LIN {X 0,Y 129.211,Z 756.744,A -85,B 0,C 180,E1 22949.999,E2 22949.999} C_VEL
LIN {X 0,Y 129.325,Z 753.398,A -85,B 0,C 180,E1 22963.541,E2 22963.541} C_VEL
LIN {X 0,Y 134.133,Z 744.964,A -85,B 0,C 180,E1 22978.668,E2 22978.668} C_VEL
LIN {X 0,Y 146.66,Z 730.342,A -85,B 0,C 180,E1 22993.136,E2 22993.136} C_VEL
LIN {X 0,Y 165.2,Z 710.054,A -85,B 0,C 180,E1 23004.51,E2 23004.51} C_VEL
LIN {X 0,Y 185.625,Z 685.738,A -85,B 0,C 180,E1 23012.504,E2 23012.504} C_VEL
LIN {X 0,Y 207.518,Z 655.091,A -85,B 0,C 180,E1 23018.501,E2 23018.501} C_VEL
LIN {X 0,Y 215.417,Z 642.118,A -85,B 0,C 180,E1 23020.306,E2 23020.306} C_VEL
LIN {X 0,Y 215.382,Z 624.11,A -85,B 0,C 180,E1 23027.832,E2 23027.832} C_VEL
LIN {X 0,Y 214.717,Z 611.173,A -85,B 0,C 180,E1 23034.95,E2 23034.95} C_VEL
LIN {X 0,Y 214.173,Z 602.579,A -85,B 0,C 180,E1 23042.032,E2 23042.032} C_VEL
LIN {X 0,Y 213.598,Z 600.314,A -85,B 0,C 180,E1 23047.07,E2 23047.07} C_VEL
LIN {X 0,Y 213.293,Z 600.443,A -85,B 0,C 180,E1 23052.301,E2 23052.301} C_VEL
LIN {X 0,Y 213.648,Z 604.341,A -85,B 0,C 180,E1 23059.613,E2 23059.613} C_VEL
LIN {X 0,Y 213.891,Z 612.007,A -85,B 0,C 180,E1 23066.156,E2 23066.156} C_VEL
LIN {X 0,Y 213.79,Z 622.244,A -85,B 0,C 180,E1 23072.194,E2 23072.194} C_VEL
LIN {X 0,Y 212.097,Z 636.594,A -85,B 0,C 180,E1 23078.779,E2 23078.779} C_VEL
LIN {X 0,Y 211.489,Z 639.855,A -85,B 0,C 180,E1 23080.121,E2 23080.121} C_VEL
LIN {X 0,Y 190.678,Z 668.162,A -85,B 0,C 180,E1 23085.989,E2 23085.989} C_VEL
LIN {X 0,Y 168.948,Z 692.69,A -85,B 0,C 180,E1 23094.372,E2 23094.372} C_VEL
LIN {X 0,Y 151.293,Z 710.245,A -85,B 0,C 180,E1 23104.541,E2 23104.541} C_VEL
LIN {X 0,Y 137.075,Z 724.356,A -85,B 0,C 180,E1 23118.856,E2 23118.856} C_VEL
LIN {X 0,Y 135.25,Z 726.254,A -85,B 0,C 180,E1 23121.71,E2 23121.71} C_VEL
LIN {X 0,Y 130.181,Z 729.523,A -85,B 0,C 180,E1 23126.752,E2 23126.752} C_VEL
LIN {X 0,Y 121.617,Z 733.742,A -85,B 0,C 180,E1 23135.865,E2 23135.865} C_VEL
LIN {X 0,Y 120.411,Z 736.776,A -85,B 0,C 180,E1 23152.164,E2 23152.164} C_VEL
LIN {X 0,Y 125.029,Z 736.093,A -85,B 0,C 180,E1 23167.267,E2 23167.267} C_VEL
LIN {X 0,Y 137.565,Z 730.863,A -85,B 0,C 180,E1 23183.419,E2 23183.419} C_VEL
LIN {X 0,Y 152.081,Z 723.611,A -85,B 0,C 180,E1 23193.645,E2 23193.645} C_VEL
LIN {X 0,Y 153.895,Z 722.33,A -85,B 0,C 180,E1 23195.406,E2 23195.406} C_VEL
LIN {X 0,Y 141.989,Z 726.974,A -85,B 0,C 180,E1 23238.646,E2 23238.646} C_VEL
LIN {X 0,Y 161.597,Z 727.84,A -85,B 0,C 180,E1 23253.222,E2 23253.222} C_VEL
LIN {X 0,Y 140.171,Z 742.415,A -85,B 0,C 180,E1 23265.602,E2 23265.602} C_VEL
LIN {X 0,Y 126.059,Z 751.755,A -85,B 0,C 180,E1 23281.284,E2 23281.284} C_VEL
LIN {X 0,Y 121.229,Z 755.582,A -85,B 0,C 180,E1 23295.533,E2 23295.533} C_VEL
LIN {X 0,Y 121.324,Z 756.048,A -85,B 0,C 180,E1 23309.999,E2 23309.999} C_VEL
LIN {X 0,Y 121.55,Z 752.592,A -85,B 0,C 180,E1 23324.425,E2 23324.425} C_VEL
LIN {X 0,Y 127.036,Z 744.011,A -85,B 0,C 180,E1 23340.433,E2 23340.433} C_VEL
LIN {X 0,Y 140.428,Z 729.533,A -85,B 0,C 180,E1 23355.218,E2 23355.218} C_VEL
LIN {X 0,Y 160.668,Z 708.594,A -85,B 0,C 180,E1 23366.99,E2 23366.99} C_VEL
LIN {X 0,Y 183.382,Z 682.398,A -85,B 0,C 180,E1 23375.26,E2 23375.26} C_VEL
LIN {X 0,Y 205.384,Z 651.952,A -85,B 0,C 180,E1 23380.85,E2 23380.85} C_VEL
LIN {X 0,Y 209.727,Z 645.118,A -85,B 0,C 180,E1 23381.778,E2 23381.778} C_VEL
LIN {X 0,Y 210.402,Z 629.378,A -85,B 0,C 180,E1 23388.669,E2 23388.669} C_VEL
LIN {X 0,Y 210.277,Z 616.843,A -85,B 0,C 180,E1 23395.877,E2 23395.877} C_VEL
LIN {X 0,Y 210.204,Z 609.566,A -85,B 0,C 180,E1 23402.07,E2 23402.07} C_VEL
LIN {X 0,Y 210.16,Z 607.952,A -85,B 0,C 180,E1 23404.138,E2 23404.138} C_VEL
LIN {X 0,Y 209.656,Z 606.988,A -85,B 0,C 180,E1 23408.311,E2 23408.311} C_VEL
LIN {X 0,Y 209.411,Z 609.111,A -85,B 0,C 180,E1 23416.816,E2 23416.816} C_VEL
LIN {X 0,Y 209.353,Z 615.396,A -85,B 0,C 180,E1 23423.535,E2 23423.535} C_VEL
LIN {X 0,Y 208.861,Z 625.795,A -85,B 0,C 180,E1 23430.5,E2 23430.5} C_VEL
LIN {X 0,Y 206.534,Z 640.522,A -85,B 0,C 180,E1 23437.677,E2 23437.677} C_VEL
LIN {X 0,Y 205.243,Z 643.906,A -85,B 0,C 180,E1 23438.832,E2 23438.832} C_VEL
LIN {X 0,Y 183.851,Z 671.424,A -85,B 0,C 180,E1 23444.741,E2 23444.741} C_VEL
LIN {X 0,Y 161.506,Z 695.254,A -85,B 0,C 180,E1 23453.299,E2 23453.299} C_VEL
LIN {X 0,Y 142.147,Z 713.441,A -85,B 0,C 180,E1 23464.783,E2 23464.783} C_VEL
LIN {X 0,Y 128.275,Z 726.429,A -85,B 0,C 180,E1 23479.803,E2 23479.803} C_VEL
LIN {X 0,Y 121.71,Z 733.639,A -85,B 0,C 180,E1 23495.532,E2 23495.532} C_VEL
LIN {X 0,Y 121.617,Z 733.742,A -85,B 0,C 180,E1 23495.865,E2 23495.865} C_VEL
LIN {X 0,Y 117.873,Z 735.563,A -85,B 0,C 180,E1 23501.829,E2 23501.829} C_VEL
LIN {X 0,Y 112.431,Z 737.343,A -85,B 0,C 180,E1 23511.341,E2 23511.341} C_VEL
LIN {X 0,Y 112.479,Z 737.388,A -85,B 0,C 180,E1 23512.466,E2 23512.466} C_VEL
LIN {X 0,Y 118.251,Z 736.645,A -85,B 0,C 180,E1 23529.81,E2 23529.81} C_VEL
LIN {X 0,Y 130.153,Z 732.236,A -85,B 0,C 180,E1 23544.524,E2 23544.524} C_VEL
LIN {X 0,Y 145.409,Z 725.234,A -85,B 0,C 180,E1 23555.377,E2 23555.377} C_VEL
LIN {X 0,Y 135.088,Z 729.989,A -85,B 0,C 180,E1 23599.637,E2 23599.637} C_VEL
LIN {X 0,Y 151.864,Z 730.982,A -85,B 0,C 180,E1 23612.831,E2 23612.831} C_VEL
LIN {X 0,Y 136.518,Z 740.791,A -85,B 0,C 180,E1 23621.701,E2 23621.701} C_VEL
LIN {X 0,Y 118.955,Z 751.235,A -85,B 0,C 180,E1 23639.392,E2 23639.392} C_VEL
LIN {X 0,Y 113.454,Z 754.966,A -85,B 0,C 180,E1 23654.518,E2 23654.518} C_VEL
LIN {X 0,Y 113.436,Z 755.352,A -85,B 0,C 180,E1 23669.999,E2 23669.999} C_VEL
LIN {X 0,Y 113.771,Z 751.782,A -85,B 0,C 180,E1 23685.435,E2 23685.435} C_VEL
LIN {X 0,Y 120.018,Z 743.052,A -85,B 0,C 180,E1 23702.418,E2 23702.418} C_VEL
LIN {X 0,Y 134.309,Z 728.782,A -85,B 0,C 180,E1 23717.454,E2 23717.454} C_VEL
LIN {X 0,Y 154.746,Z 708.903,A -85,B 0,C 180,E1 23728.885,E2 23728.885} C_VEL
LIN {X 0,Y 178.569,Z 682.655,A -85,B 0,C 180,E1 23737.234,E2 23737.234} C_VEL
LIN {X 0,Y 200.945,Z 652.949,A -85,B 0,C 180,E1 23742.672,E2 23742.672} C_VEL
LIN {X 0,Y 204.339,Z 647.359,A -85,B 0,C 180,E1 23743.549,E2 23743.549} C_VEL
LIN {X 0,Y 205.578,Z 630.818,A -85,B 0,C 180,E1 23751.536,E2 23751.536} C_VEL
LIN {X 0,Y 205.901,Z 619.773,A -85,B 0,C 180,E1 23758.953,E2 23758.953} C_VEL
LIN {X 0,Y 206.078,Z 614.812,A -85,B 0,C 180,E1 23764.22,E2 23764.22} C_VEL
LIN {X 0,Y 205.567,Z 613.797,A -85,B 0,C 180,E1 23768.477,E2 23768.477} C_VEL
LIN {X 0,Y 205.123,Z 616.152,A -85,B 0,C 180,E1 23777.179,E2 23777.179} C_VEL
LIN {X 0,Y 204.701,Z 621.867,A -85,B 0,C 180,E1 23783.301,E2 23783.301} C_VEL
LIN {X 0,Y 203.826,Z 630.656,A -85,B 0,C 180,E1 23789.436,E2 23789.436} C_VEL
LIN {X 0,Y 201.12,Z 643.929,A -85,B 0,C 180,E1 23796.299,E2 23796.299} C_VEL
LIN {X 0,Y 199.022,Z 647.826,A -85,B 0,C 180,E1 23797.438,E2 23797.438} C_VEL
LIN {X 0,Y 175.722,Z 676.115,A -85,B 0,C 180,E1 23803.811,E2 23803.811} C_VEL
LIN {X 0,Y 152.955,Z 698.884,A -85,B 0,C 180,E1 23812.677,E2 23812.677} C_VEL
LIN {X 0,Y 133.317,Z 716.185,A -85,B 0,C 180,E1 23824.794,E2 23824.794} C_VEL
LIN {X 0,Y 120.512,Z 727.441,A -85,B 0,C 180,E1 23839.138,E2 23839.138} C_VEL
LIN {X 0,Y 113.754,Z 734.314,A -85,B 0,C 180,E1 23855.316,E2 23855.316} C_VEL
LIN {X 0,Y 112.479,Z 737.388,A -85,B 0,C 180,E1 23872.466,E2 23872.466} C_VEL
LIN {X 0,Y 111.272,Z 737.849,A -85,B 0,C 180,E1 23879.16,E2 23879.16} C_VEL
LIN {X 0,Y 110.28,Z 737.598,A -85,B 0,C 180,E1 23890.32,E2 23890.32} C_VEL
LIN {X 0,Y 110.434,Z 737.451,A -85,B 0,C 180,E1 23890.596,E2 23890.596} C_VEL
LIN {X 0,Y 125.199,Z 732.625,A -85,B 0,C 180,E1 23907.841,E2 23907.841} C_VEL
LIN {X 0,Y 134.431,Z 728.888,A -85,B 0,C 180,E1 23914.299,E2 23914.299} C_VEL
LIN {X 0,Y 135.931,Z 727.975,A -85,B 0,C 180,E1 23916.094,E2 23916.094} C_VEL
LIN {X 0,Y 128.184,Z 732.812,A -85,B 0,C 180,E1 23960.742,E2 23960.742} C_VEL
LIN {X 0,Y 141.844,Z 733.834,A -85,B 0,C 180,E1 23972.244,E2 23972.244} C_VEL
LIN {X 0,Y 138.06,Z 736.573,A -85,B 0,C 180,E1 23975.081,E2 23975.081} C_VEL
LIN {X 0,Y 116.47,Z 748.265,A -85,B 0,C 180,E1 23991.237,E2 23991.237} C_VEL
LIN {X 0,Y 108.081,Z 752.904,A -85,B 0,C 180,E1 24005.147,E2 24005.147} C_VEL
LIN {X 0,Y 104.972,Z 754.908,A -85,B 0,C 180,E1 24021.705,E2 24021.705} C_VEL
LIN {X 0,Y 105.55,Z 754.655,A -85,B 0,C 180,E1 24029.999,E2 24029.999} C_VEL
LIN {X 0,Y 106.023,Z 750.972,A -85,B 0,C 180,E1 24046.594,E2 24046.594} C_VEL
LIN {X 0,Y 113.91,Z 741.386,A -85,B 0,C 180,E1 24065.672,E2 24065.672} C_VEL
LIN {X 0,Y 130.89,Z 725.814,A -85,B 0,C 180,E1 24081.523,E2 24081.523} C_VEL
LIN {X 0,Y 153.373,Z 704.782,A -85,B 0,C 180,E1 24092.682,E2 24092.682} C_VEL
LIN {X 0,Y 177.085,Z 679.176,A -85,B 0,C 180,E1 24100.137,E2 24100.137} C_VEL
LIN {X 0,Y 198.313,Z 651.525,A -85,B 0,C 180,E1 24104.9,E2 24104.9} C_VEL
LIN {X 0,Y 200.088,Z 641.154,A -85,B 0,C 180,E1 24109.651,E2 24109.651} C_VEL
LIN {X 0,Y 201.062,Z 629.435,A -85,B 0,C 180,E1 24116.769,E2 24116.769} C_VEL
LIN {X 0,Y 201.677,Z 623.216,A -85,B 0,C 180,E1 24122.158,E2 24122.158} C_VEL
LIN {X 0,Y 201.796,Z 621.527,A -85,B 0,C 180,E1 24124.309,E2 24124.309} C_VEL
LIN {X 0,Y 200.935,Z 620.83,A -85,B 0,C 180,E1 24131.598,E2 24131.598} C_VEL
LIN {X 0,Y 200.66,Z 623.111,A -85,B 0,C 180,E1 24137.573,E2 24137.573} C_VEL
LIN {X 0,Y 199.633,Z 629.955,A -85,B 0,C 180,E1 24144.477,E2 24144.477} C_VEL
LIN {X 0,Y 197.801,Z 639.804,A -85,B 0,C 180,E1 24150.875,E2 24150.875} C_VEL
LIN {X 0,Y 194.972,Z 649.025,A -85,B 0,C 180,E1 24155.496,E2 24155.496} C_VEL
LIN {X 0,Y 171.845,Z 676.283,A -85,B 0,C 180,E1 24161.503,E2 24161.503} C_VEL
LIN {X 0,Y 148.045,Z 699.176,A -85,B 0,C 180,E1 24170.268,E2 24170.268} C_VEL
LIN {X 0,Y 126.272,Z 717.349,A -85,B 0,C 180,E1 24183.28,E2 24183.28} C_VEL
LIN {X 0,Y 112.783,Z 728.445,A -85,B 0,C 180,E1 24198.384,E2 24198.384} C_VEL
LIN {X 0,Y 106.235,Z 734.662,A -85,B 0,C 180,E1 24213.779,E2 24213.779} C_VEL
LIN {X 0,Y 104.541,Z 737.946,A -85,B 0,C 180,E1 24232.755,E2 24232.755} C_VEL
LIN {X 0,Y 110.434,Z 737.451,A -85,B 0,C 180,E1 24250.596,E2 24250.596} C_VEL
LIN {X 0,Y 112.215,Z 736.71,A -85,B 0,C 180,E1 24257.247,E2 24257.247} C_VEL
LIN {X 0,Y 115.432,Z 734.859,A -85,B 0,C 180,E1 24267.05,E2 24267.05} C_VEL
LIN {X 0,Y 116.42,Z 734.493,A -85,B 0,C 180,E1 24268.006,E2 24268.006} C_VEL
LIN {X 0,Y 127.417,Z 730.453,A -85,B 0,C 180,E1 24276.089,E2 24276.089} C_VEL
LIN {X 0,Y 121.255,Z 735.402,A -85,B 0,C 180,E1 24321.987,E2 24321.987} C_VEL
LIN {X 0,Y 132.231,Z 736.354,A -85,B 0,C 180,E1 24331.735,E2 24331.735} C_VEL
LIN {X 0,Y 128.797,Z 738.699,A -85,B 0,C 180,E1 24334.621,E2 24334.621} C_VEL
LIN {X 0,Y 107.387,Z 749.098,A -85,B 0,C 180,E1 24351.887,E2 24351.887} C_VEL
LIN {X 0,Y 98.025,Z 753.726,A -85,B 0,C 180,E1 24372.004,E2 24372.004} C_VEL
LIN {X 0,Y 97.656,Z 753.958,A -85,B 0,C 180,E1 24389.998,E2 24389.998} C_VEL
LIN {X 0,Y 98.319,Z 750.158,A -85,B 0,C 180,E1 24407.937,E2 24407.937} C_VEL
LIN {X 0,Y 107.14,Z 740.567,A -85,B 0,C 180,E1 24427.98,E2 24427.98} C_VEL
LIN {X 0,Y 126.193,Z 724.413,A -85,B 0,C 180,E1 24444.629,E2 24444.629} C_VEL
LIN {X 0,Y 149.737,Z 703.397,A -85,B 0,C 180,E1 24455.512,E2 24455.512} C_VEL
LIN {X 0,Y 174.454,Z 677.594,A -85,B 0,C 180,E1 24462.687,E2 24462.687} C_VEL
LIN {X 0,Y 192.924,Z 654.338,A -85,B 0,C 180,E1 24466.605,E2 24466.605} C_VEL
LIN {X 0,Y 194.91,Z 645.123,A -85,B 0,C 180,E1 24471.07,E2 24471.07} C_VEL
LIN {X 0,Y 196.559,Z 633.429,A -85,B 0,C 180,E1 24478.903,E2 24478.903} C_VEL
LIN {X 0,Y 197.249,Z 628.079,A -85,B 0,C 180,E1 24484.409,E2 24484.409} C_VEL
LIN {X 0,Y 196.878,Z 627.081,A -85,B 0,C 180,E1 24488.854,E2 24488.854} C_VEL
LIN {X 0,Y 196.133,Z 628.593,A -85,B 0,C 180,E1 24495.682,E2 24495.682} C_VEL
LIN {X 0,Y 195.291,Z 633.054,A -85,B 0,C 180,E1 24501.509,E2 24501.509} C_VEL
LIN {X 0,Y 193.357,Z 641.473,A -85,B 0,C 180,E1 24508.03,E2 24508.03} C_VEL
LIN {X 0,Y 190.363,Z 651.076,A -85,B 0,C 180,E1 24513.546,E2 24513.546} C_VEL
LIN {X 0,Y 166.365,Z 678.32,A -85,B 0,C 180,E1 24519.624,E2 24519.624} C_VEL
LIN {X 0,Y 141.655,Z 700.963,A -85,B 0,C 180,E1 24528.474,E2 24528.474} C_VEL
LIN {X 0,Y 119.326,Z 718.509,A -85,B 0,C 180,E1 24541.588,E2 24541.588} C_VEL
LIN {X 0,Y 105.073,Z 729.441,A -85,B 0,C 180,E1 24557.518,E2 24557.518} C_VEL
LIN {X 0,Y 98.152,Z 735.516,A -85,B 0,C 180,E1 24574.091,E2 24574.091} C_VEL
LIN {X 0,Y 96.394,Z 738.324,A -85,B 0,C 180,E1 24589.502,E2 24589.502} C_VEL
LIN {X 0,Y 100.543,Z 738.777,A -85,B 0,C 180,E1 24607.042,E2 24607.042} C_VEL
LIN {X 0,Y 112.23,Z 735.889,A -85,B 0,C 180,E1 24624.046,E2 24624.046} C_VEL
LIN {X 0,Y 116.42,Z 734.493,A -85,B 0,C 180,E1 24628.006,E2 24628.006} C_VEL
LIN {X 0,Y 118.537,Z 733.336,A -85,B 0,C 180,E1 24632.951,E2 24632.951} C_VEL
LIN {X 0,Y 116.54,Z 733.107,A -85,B 0,C 180,E1 24638.161,E2 24638.161} C_VEL
LIN {X 0,Y 115.413,Z 733.231,A -85,B 0,C 180,E1 24639.607,E2 24639.607} C_VEL
LIN {X 0,Y 121,Z 738.501,A -85,B 0,C 180,E1 24690.02,E2 24690.02} C_VEL
LIN {X 0,Y 122.539,Z 738.617,A -85,B 0,C 180,E1 24691.188,E2 24691.188} C_VEL
LIN {X 0,Y 120.942,Z 739.886,A -85,B 0,C 180,E1 24693.287,E2 24693.287} C_VEL
LIN {X 0,Y 98.65,Z 749.589,A -85,B 0,C 180,E1 24712.123,E2 24712.123} C_VEL
LIN {X 0,Y 90.414,Z 753.081,A -85,B 0,C 180,E1 24730.43,E2 24730.43} C_VEL
LIN {X 0,Y 89.754,Z 753.248,A -85,B 0,C 180,E1 24749.998,E2 24749.998} C_VEL
LIN {X 0,Y 90.689,Z 749.321,A -85,B 0,C 180,E1 24769.505,E2 24769.505} C_VEL
LIN {X 0,Y 100.07,Z 740.157,A -85,B 0,C 180,E1 24789.915,E2 24789.915} C_VEL
LIN {X 0,Y 119.859,Z 724.599,A -85,B 0,C 180,E1 24806.812,E2 24806.812} C_VEL
LIN {X 0,Y 144.965,Z 703.441,A -85,B 0,C 180,E1 24817.964,E2 24817.964} C_VEL
LIN {X 0,Y 170.781,Z 677.579,A -85,B 0,C 180,E1 24825.016,E2 24825.016} C_VEL
LIN {X 0,Y 188.051,Z 656.751,A -85,B 0,C 180,E1 24828.464,E2 24828.464} C_VEL
LIN {X 0,Y 190.704,Z 644.606,A -85,B 0,C 180,E1 24835.453,E2 24835.453} C_VEL
LIN {X 0,Y 192.352,Z 635.585,A -85,B 0,C 180,E1 24843.124,E2 24843.124} C_VEL
LIN {X 0,Y 192.176,Z 633.525,A -85,B 0,C 180,E1 24849.073,E2 24849.073} C_VEL
LIN {X 0,Y 191.22,Z 635.469,A -85,B 0,C 180,E1 24856.552,E2 24856.552} C_VEL
LIN {X 0,Y 189.475,Z 641.763,A -85,B 0,C 180,E1 24863.556,E2 24863.556} C_VEL
LIN {X 0,Y 186.092,Z 651.832,A -85,B 0,C 180,E1 24870.452,E2 24870.452} C_VEL
LIN {X 0,Y 184.979,Z 654.533,A -85,B 0,C 180,E1 24871.9,E2 24871.9} C_VEL
LIN {X 0,Y 160.123,Z 681.223,A -85,B 0,C 180,E1 24877.878,E2 24877.878} C_VEL
LIN {X 0,Y 135.895,Z 702.342,A -85,B 0,C 180,E1 24886.287,E2 24886.287} C_VEL
LIN {X 0,Y 112.484,Z 719.661,A -85,B 0,C 180,E1 24899.685,E2 24899.685} C_VEL
LIN {X 0,Y 97.367,Z 730.431,A -85,B 0,C 180,E1 24916.513,E2 24916.513} C_VEL
LIN {X 0,Y 90.896,Z 735.686,A -85,B 0,C 180,E1 24931.521,E2 24931.521} C_VEL
LIN {X 0,Y 88.535,Z 738.945,A -85,B 0,C 180,E1 24950.003,E2 24950.003} C_VEL
LIN {X 0,Y 93.841,Z 739.388,A -85,B 0,C 180,E1 24970.198,E2 24970.198} C_VEL
LIN {X 0,Y 109.782,Z 735.547,A -85,B 0,C 180,E1 24990.111,E2 24990.111} C_VEL
LIN {X 0,Y 116.722,Z 733.41,A -85,B 0,C 180,E1 24995.239,E2 24995.239} C_VEL
LIN {X 0,Y 117.6,Z 732.943,A -85,B 0,C 180,E1 24997.268,E2 24997.268} C_VEL
LIN {X 0,Y 115.413,Z 733.231,A -85,B 0,C 180,E1 24999.607,E2 24999.607} C_VEL
LIN {X 0,Y 106.139,Z 735.188,A -85,B 0,C 180,E1 25007.212,E2 25007.212} C_VEL
LIN {X 0,Y 99.236,Z 737.09,A -85,B 0,C 180,E1 25016.092,E2 25016.092} C_VEL
LIN {X 0,Y 113.376,Z 740.648,A -85,B 0,C 180,E1 25050.961,E2 25050.961} C_VEL
LIN {X 0,Y 104.612,Z 744.424,A -85,B 0,C 180,E1 25057.243,E2 25057.243} C_VEL
LIN {X 0,Y 86.571,Z 751.161,A -85,B 0,C 180,E1 25078.35,E2 25078.35} C_VEL
LIN {X 0,Y 81.343,Z 752.887,A -85,B 0,C 180,E1 25099.27,E2 25099.27} C_VEL
LIN {X 0,Y 81.851,Z 752.515,A -85,B 0,C 180,E1 25109.998,E2 25109.998} C_VEL
LIN {X 0,Y 83.122,Z 748.464,A -85,B 0,C 180,E1 25131.363,E2 25131.363} C_VEL
LIN {X 0,Y 93.913,Z 739.159,A -85,B 0,C 180,E1 25153.134,E2 25153.134} C_VEL
LIN {X 0,Y 115.531,Z 723.433,A -85,B 0,C 180,E1 25170.253,E2 25170.253} C_VEL
LIN {X 0,Y 142.085,Z 702.095,A -85,B 0,C 180,E1 25181.039,E2 25181.039} C_VEL
LIN {X 0,Y 168.814,Z 675.895,A -85,B 0,C 180,E1 25187.757,E2 25187.757} C_VEL
LIN {X 0,Y 183.076,Z 659.092,A -85,B 0,C 180,E1 25190.487,E2 25190.487} C_VEL
LIN {X 0,Y 185.92,Z 648.006,A -85,B 0,C 180,E1 25197.674,E2 25197.674} C_VEL
LIN {X 0,Y 187.673,Z 640.866,A -85,B 0,C 180,E1 25204.634,E2 25204.634} C_VEL
LIN {X 0,Y 187.319,Z 639.833,A -85,B 0,C 180,E1 25209.31,E2 25209.31} C_VEL
LIN {X 0,Y 186.164,Z 642.022,A -85,B 0,C 180,E1 25217.015,E2 25217.015} C_VEL
LIN {X 0,Y 183.639,Z 648.995,A -85,B 0,C 180,E1 25224.353,E2 25224.353} C_VEL
LIN {X 0,Y 180.042,Z 657.518,A -85,B 0,C 180,E1 25230.003,E2 25230.003} C_VEL
LIN {X 0,Y 154.289,Z 683.851,A -85,B 0,C 180,E1 25235.944,E2 25235.944} C_VEL
LIN {X 0,Y 128.127,Z 705.333,A -85,B 0,C 180,E1 25244.845,E2 25244.845} C_VEL
LIN {X 0,Y 103.657,Z 722.251,A -85,B 0,C 180,E1 25259.255,E2 25259.255} C_VEL
LIN {X 0,Y 87.243,Z 733.154,A -85,B 0,C 180,E1 25280.007,E2 25280.007} C_VEL
LIN {X 0,Y 80.886,Z 738.321,A -85,B 0,C 180,E1 25300.791,E2 25300.791} C_VEL
LIN {X 0,Y 82.966,Z 740.306,A -85,B 0,C 180,E1 25323.198,E2 25323.198} C_VEL
LIN {X 0,Y 94.157,Z 738.906,A -85,B 0,C 180,E1 25343.52,E2 25343.52} C_VEL
LIN {X 0,Y 106.144,Z 735.95,A -85,B 0,C 180,E1 25354.651,E2 25354.651} C_VEL
LIN {X 0,Y 108.466,Z 735.101,A -85,B 0,C 180,E1 25357.955,E2 25357.955} C_VEL
LIN {X 0,Y 99.236,Z 737.09,A -85,B 0,C 180,E1 25376.092,E2 25376.092} C_VEL
LIN {X 0,Y 94.999,Z 739.005,A -85,B 0,C 180,E1 25386.08,E2 25386.08} C_VEL
LIN {X 0,Y 93.905,Z 740.923,A -85,B 0,C 180,E1 25396.638,E2 25396.638} C_VEL
LIN {X 0,Y 104.139,Z 742.372,A -85,B 0,C 180,E1 25410.572,E2 25410.572} C_VEL
LIN {X 0,Y 82.743,Z 749.641,A -85,B 0,C 180,E1 25430.171,E2 25430.171} C_VEL
LIN {X 0,Y 73.511,Z 752.212,A -85,B 0,C 180,E1 25458.112,E2 25458.112} C_VEL
LIN {X 0,Y 73.947,Z 751.779,A -85,B 0,C 180,E1 25469.998,E2 25469.998} C_VEL
LIN {X 0,Y 75.645,Z 747.602,A -85,B 0,C 180,E1 25493.596,E2 25493.596} C_VEL
LIN {X 0,Y 88.742,Z 737.729,A -85,B 0,C 180,E1 25517.533,E2 25517.533} C_VEL
LIN {X 0,Y 113.082,Z 721.247,A -85,B 0,C 180,E1 25534.659,E2 25534.659} C_VEL
LIN {X 0,Y 141.256,Z 699.246,A -85,B 0,C 180,E1 25544.729,E2 25544.729} C_VEL
LIN {X 0,Y 168.719,Z 672.61,A -85,B 0,C 180,E1 25550.803,E2 25550.803} C_VEL
LIN {X 0,Y 178.097,Z 661.699,A -85,B 0,C 180,E1 25552.691,E2 25552.691} C_VEL
LIN {X 0,Y 181.242,Z 651.538,A -85,B 0,C 180,E1 25560.007,E2 25560.007} C_VEL
LIN {X 0,Y 182.557,Z 646.82,A -85,B 0,C 180,E1 25565.58,E2 25565.58} C_VEL
LIN {X 0,Y 182.281,Z 646.039,A -85,B 0,C 180,E1 25569.57,E2 25569.57} C_VEL
LIN {X 0,Y 180.97,Z 648.251,A -85,B 0,C 180,E1 25577.034,E2 25577.034} C_VEL
LIN {X 0,Y 177.869,Z 655.178,A -85,B 0,C 180,E1 25584.349,E2 25584.349} C_VEL
LIN {X 0,Y 175.009,Z 660.687,A -85,B 0,C 180,E1 25588.065,E2 25588.065} C_VEL
LIN {X 0,Y 148.296,Z 686.781,A -85,B 0,C 180,E1 25593.947,E2 25593.947} C_VEL
LIN {X 0,Y 122.738,Z 706.609,A -85,B 0,C 180,E1 25602.256,E2 25602.256} C_VEL
LIN {X 0,Y 96.985,Z 723.35,A -85,B 0,C 180,E1 25616.881,E2 25616.881} C_VEL
LIN {X 0,Y 79.442,Z 734.09,A -85,B 0,C 180,E1 25639.015,E2 25639.015} C_VEL
LIN {X 0,Y 72.839,Z 739.126,A -85,B 0,C 180,E1 25662,E2 25662} C_VEL
LIN {X 0,Y 76.171,Z 740.971,A -85,B 0,C 180,E1 25687.311,E2 25687.311} C_VEL
LIN {X 0,Y 91.273,Z 739.009,A -85,B 0,C 180,E1 25710.14,E2 25710.14} C_VEL
LIN {X 0,Y 98.98,Z 737.285,A -85,B 0,C 180,E1 25716.615,E2 25716.615} C_VEL
LIN {X 0,Y 99.756,Z 737.054,A -85,B 0,C 180,E1 25718.204,E2 25718.204} C_VEL
LIN {X 0,Y 93.905,Z 740.923,A -85,B 0,C 180,E1 25756.638,E2 25756.638} C_VEL
LIN {X 0,Y 94.939,Z 742.293,A -85,B 0,C 180,E1 25763.988,E2 25763.988} C_VEL
LIN {X 0,Y 92.163,Z 744.389,A -85,B 0,C 180,E1 25770.616,E2 25770.616} C_VEL
LIN {X 0,Y 91.816,Z 744.493,A -85,B 0,C 180,E1 25771.027,E2 25771.027} C_VEL
LIN {X 0,Y 76.661,Z 749.066,A -85,B 0,C 180,E1 25786.266,E2 25786.266} C_VEL
LIN {X 0,Y 65.689,Z 751.535,A -85,B 0,C 180,E1 25816.671,E2 25816.671} C_VEL
LIN {X 0,Y 66.033,Z 751.042,A -85,B 0,C 180,E1 25829.998,E2 25829.998} C_VEL
LIN {X 0,Y 68.297,Z 746.739,A -85,B 0,C 180,E1 25856.318,E2 25856.318} C_VEL
LIN {X 0,Y 82.215,Z 737.418,A -85,B 0,C 180,E1 25880.521,E2 25880.521} C_VEL
LIN {X 0,Y 108.256,Z 721.028,A -85,B 0,C 180,E1 25897.907,E2 25897.907} C_VEL
LIN {X 0,Y 137.08,Z 699.634,A -85,B 0,C 180,E1 25907.471,E2 25907.471} C_VEL
LIN {X 0,Y 165.262,Z 673.422,A -85,B 0,C 180,E1 25913.223,E2 25913.223} C_VEL
LIN {X 0,Y 172.941,Z 664.907,A -85,B 0,C 180,E1 25914.577,E2 25914.577} C_VEL
LIN {X 0,Y 176.276,Z 656.026,A -85,B 0,C 180,E1 25921.629,E2 25921.629} C_VEL
LIN {X 0,Y 177.333,Z 653.105,A -85,B 0,C 180,E1 25924.905,E2 25924.905} C_VEL
LIN {X 0,Y 177.062,Z 652.138,A -85,B 0,C 180,E1 25929.854,E2 25929.854} C_VEL
LIN {X 0,Y 176.029,Z 653.233,A -85,B 0,C 180,E1 25934.961,E2 25934.961} C_VEL
LIN {X 0,Y 173.548,Z 657.993,A -85,B 0,C 180,E1 25941.418,E2 25941.418} C_VEL
LIN {X 0,Y 169.983,Z 664.026,A -85,B 0,C 180,E1 25946.037,E2 25946.037} C_VEL
LIN {X 0,Y 142.488,Z 689.555,A -85,B 0,C 180,E1 25951.779,E2 25951.779} C_VEL
LIN {X 0,Y 114.694,Z 709.871,A -85,B 0,C 180,E1 25960.619,E2 25960.619} C_VEL
LIN {X 0,Y 88.176,Z 725.701,A -85,B 0,C 180,E1 25976.079,E2 25976.079} C_VEL
LIN {X 0,Y 71.654,Z 735.016,A -85,B 0,C 180,E1 25997.803,E2 25997.803} C_VEL
LIN {X 0,Y 64.789,Z 739.929,A -85,B 0,C 180,E1 26023.517,E2 26023.517} C_VEL
LIN {X 0,Y 69.314,Z 741.646,A -85,B 0,C 180,E1 26050.947,E2 26050.947} C_VEL
LIN {X 0,Y 87.211,Z 739.54,A -85,B 0,C 180,E1 26075.182,E2 26075.182} C_VEL
LIN {X 0,Y 91.053,Z 738.797,A -85,B 0,C 180,E1 26078.443,E2 26078.443} C_VEL
LIN {X 0,Y 93.718,Z 743.71,A -85,B 0,C 180,E1 26128.973,E2 26128.973} C_VEL
LIN {X 0,Y 91.816,Z 744.493,A -85,B 0,C 180,E1 26131.027,E2 26131.027} C_VEL
LIN {X 0,Y 86.319,Z 746.19,A -85,B 0,C 180,E1 26135.154,E2 26135.154} C_VEL
LIN {X 0,Y 67.442,Z 749.319,A -85,B 0,C 180,E1 26146.793,E2 26146.793} C_VEL
LIN {X 0,Y 66.27,Z 749.486,A -85,B 0,C 180,E1 26148.429,E2 26148.429} C_VEL
LIN {X 0,Y 57.911,Z 750.857,A -85,B 0,C 180,E1 26174.841,E2 26174.841} C_VEL
LIN {X 0,Y 58.103,Z 750.295,A -85,B 0,C 180,E1 26189.997,E2 26189.997} C_VEL
LIN {X 0,Y 61.155,Z 745.856,A -85,B 0,C 180,E1 26219.678,E2 26219.678} C_VEL
LIN {X 0,Y 77.833,Z 736.079,A -85,B 0,C 180,E1 26245.764,E2 26245.764} C_VEL
LIN {X 0,Y 105.424,Z 719.805,A -85,B 0,C 180,E1 26262.076,E2 26262.076} C_VEL
LIN {X 0,Y 135.512,Z 698.197,A -85,B 0,C 180,E1 26270.932,E2 26270.932} C_VEL
LIN {X 0,Y 165.046,Z 671.159,A -85,B 0,C 180,E1 26276.174,E2 26276.174} C_VEL
LIN {X 0,Y 168.112,Z 667.714,A -85,B 0,C 180,E1 26276.891,E2 26276.891} C_VEL
LIN {X 0,Y 171.441,Z 659.965,A -85,B 0,C 180,E1 26283.805,E2 26283.805} C_VEL
LIN {X 0,Y 171.858,Z 658.989,A -85,B 0,C 180,E1 26285.062,E2 26285.062} C_VEL
LIN {X 0,Y 171.588,Z 658.068,A -85,B 0,C 180,E1 26290.172,E2 26290.172} C_VEL
LIN {X 0,Y 169.784,Z 660.266,A -85,B 0,C 180,E1 26297.047,E2 26297.047} C_VEL
LIN {X 0,Y 166.825,Z 665.187,A -85,B 0,C 180,E1 26302.584,E2 26302.584} C_VEL
LIN {X 0,Y 165.53,Z 667.014,A -85,B 0,C 180,E1 26303.838,E2 26303.838} C_VEL
LIN {X 0,Y 136.89,Z 692.3,A -85,B 0,C 180,E1 26309.422,E2 26309.422} C_VEL
LIN {X 0,Y 106.727,Z 712.967,A -85,B 0,C 180,E1 26318.716,E2 26318.716} C_VEL
LIN {X 0,Y 79.34,Z 728.058,A -85,B 0,C 180,E1 26335.077,E2 26335.077} C_VEL
LIN {X 0,Y 63.882,Z 735.941,A -85,B 0,C 180,E1 26356.292,E2 26356.292} C_VEL
LIN {X 0,Y 56.818,Z 740.729,A -85,B 0,C 180,E1 26385.458,E2 26385.458} C_VEL
LIN {X 0,Y 63.096,Z 742.318,A -85,B 0,C 180,E1 26416.05,E2 26416.05} C_VEL
LIN {X 0,Y 81.281,Z 740.491,A -85,B 0,C 180,E1 26438.662,E2 26438.662} C_VEL
LIN {X 0,Y 84.131,Z 745.013,A -85,B 0,C 180,E1 26488.605,E2 26488.605} C_VEL
LIN {X 0,Y 80.57,Z 746.184,A -85,B 0,C 180,E1 26492.253,E2 26492.253} C_VEL
LIN {X 0,Y 66.27,Z 749.486,A -85,B 0,C 180,E1 26508.429,E2 26508.429} C_VEL
LIN {X 0,Y 58.834,Z 750.292,A -85,B 0,C 180,E1 26518.333,E2 26518.333} C_VEL
LIN {X 0,Y 49.624,Z 749.906,A -85,B 0,C 180,E1 26539.704,E2 26539.704} C_VEL
LIN {X 0,Y 50.175,Z 749.547,A -85,B 0,C 180,E1 26549.997,E2 26549.997} C_VEL
LIN {X 0,Y 53.725,Z 745.314,A -85,B 0,C 180,E1 26582.329,E2 26582.329} C_VEL
LIN {X 0,Y 73.512,Z 735.047,A -85,B 0,C 180,E1 26611.084,E2 26611.084} C_VEL
LIN {X 0,Y 103.184,Z 718.586,A -85,B 0,C 180,E1 26626.439,E2 26626.439} C_VEL
LIN {X 0,Y 134.581,Z 696.67,A -85,B 0,C 180,E1 26634.458,E2 26634.458} C_VEL
LIN {X 0,Y 163.157,Z 670.951,A -85,B 0,C 180,E1 26639.006,E2 26639.006} C_VEL
LIN {X 0,Y 166.238,Z 664.748,A -85,B 0,C 180,E1 26645.233,E2 26645.233} C_VEL
LIN {X 0,Y 165.959,Z 663.847,A -85,B 0,C 180,E1 26650.521,E2 26650.521} C_VEL
LIN {X 0,Y 163.709,Z 666.432,A -85,B 0,C 180,E1 26657.532,E2 26657.532} C_VEL
LIN {X 0,Y 160.797,Z 670.426,A -85,B 0,C 180,E1 26661.59,E2 26661.59} C_VEL
LIN {X 0,Y 131.551,Z 695.04,A -85,B 0,C 180,E1 26666.877,E2 26666.877} C_VEL
LIN {X 0,Y 102.024,Z 714.195,A -85,B 0,C 180,E1 26675.292,E2 26675.292} C_VEL
LIN {X 0,Y 73.028,Z 729.091,A -85,B 0,C 180,E1 26691.54,E2 26691.54} C_VEL
LIN {X 0,Y 56.137,Z 736.869,A -85,B 0,C 180,E1 26714.355,E2 26714.355} C_VEL
LIN {X 0,Y 48.864,Z 741.536,A -85,B 0,C 180,E1 26748.055,E2 26748.055} C_VEL
LIN {X 0,Y 57.471,Z 742.992,A -85,B 0,C 180,E1 26782.224,E2 26782.224} C_VEL
LIN {X 0,Y 72.253,Z 741.901,A -85,B 0,C 180,E1 26800.3,E2 26800.3} C_VEL
LIN {X 0,Y 74.597,Z 745.811,A -85,B 0,C 180,E1 26846.76,E2 26846.76} C_VEL
LIN {X 0,Y 70.932,Z 746.912,A -85,B 0,C 180,E1 26851.364,E2 26851.364} C_VEL
LIN {X 0,Y 53.153,Z 749.987,A -85,B 0,C 180,E1 26878.658,E2 26878.658} C_VEL
LIN {X 0,Y 49.624,Z 749.906,A -85,B 0,C 180,E1 26899.704,E2 26899.704} C_VEL
LIN {X 0,Y 46.928,Z 749.302,A -85,B 0,C 180,E1 26909.431,E2 26909.431} C_VEL
LIN {X 0,Y 42.555,Z 747.239,A -85,B 0,C 180,E1 26927.917,E2 26927.917} C_VEL
LIN {X 0,Y 56.069,Z 740.278,A -85,B 0,C 180,E1 26964.104,E2 26964.104} C_VEL
LIN {X 0,Y 83.978,Z 727.054,A -85,B 0,C 180,E1 26984.819,E2 26984.819} C_VEL
LIN {X 0,Y 115.963,Z 708.276,A -85,B 0,C 180,E1 26994.602,E2 26994.602} C_VEL
LIN {X 0,Y 148.033,Z 683.586,A -85,B 0,C 180,E1 27000.009,E2 27000.009} C_VEL
LIN {X 0,Y 158.381,Z 673.853,A -85,B 0,C 180,E1 27001.623,E2 27001.623} C_VEL
LIN {X 0,Y 160.449,Z 670.392,A -85,B 0,C 180,E1 27005.423,E2 27005.423} C_VEL
LIN {X 0,Y 160.091,Z 669.556,A -85,B 0,C 180,E1 27010.911,E2 27010.911} C_VEL
LIN {X 0,Y 158.126,Z 671.59,A -85,B 0,C 180,E1 27016.76,E2 27016.76} C_VEL
LIN {X 0,Y 157.053,Z 672.85,A -85,B 0,C 180,E1 27018.508,E2 27018.508} C_VEL
LIN {X 0,Y 152.774,Z 676.878,A -85,B 0,C 180,E1 27019.693,E2 27019.693} C_VEL
LIN {X 0,Y 123.027,Z 700.001,A -85,B 0,C 180,E1 27024.82,E2 27024.82} C_VEL
LIN {X 0,Y 91.218,Z 718.862,A -85,B 0,C 180,E1 27033.91,E2 27033.91} C_VEL
LIN {X 0,Y 61.734,Z 732.336,A -85,B 0,C 180,E1 27052.185,E2 27052.185} C_VEL
LIN {X 0,Y 44.865,Z 739.326,A -85,B 0,C 180,E1 27081.33,E2 27081.33} C_VEL
LIN {X 0,Y 41.072,Z 742.341,A -85,B 0,C 180,E1 27111.637,E2 27111.637} C_VEL
LIN {X 0,Y 56.119,Z 743.564,A -85,B 0,C 180,E1 27154.292,E2 27154.292} C_VEL
LIN {X 0,Y 63.124,Z 743.172,A -85,B 0,C 180,E1 27162.89,E2 27162.89} C_VEL
LIN {X 0,Y 64.596,Z 746.399,A -85,B 0,C 180,E1 27204.193,E2 27204.193} C_VEL
LIN {X 0,Y 64.508,Z 746.8,A -85,B 0,C 180,E1 27207.357,E2 27207.357} C_VEL
LIN {X 0,Y 47.549,Z 749.204,A -85,B 0,C 180,E1 27230.438,E2 27230.438} C_VEL
LIN {X 0,Y 42.244,Z 748.8,A -85,B 0,C 180,E1 27269.996,E2 27269.996} C_VEL
LIN {X 0,Y 42.555,Z 747.239,A -85,B 0,C 180,E1 27287.917,E2 27287.917} C_VEL
LIN {X 0,Y 43.65,Z 745.045,A -85,B 0,C 180,E1 27305.054,E2 27305.054} C_VEL
LIN {X 0,Y 49.141,Z 740.324,A -85,B 0,C 180,E1 27328.3,E2 27328.3} C_VEL
LIN {X 0,Y 50.549,Z 739.746,A -85,B 0,C 180,E1 27330.162,E2 27330.162} C_VEL
LIN {X 0,Y 80.455,Z 726.753,A -85,B 0,C 180,E1 27349.756,E2 27349.756} C_VEL
LIN {X 0,Y 113.602,Z 708.12,A -85,B 0,C 180,E1 27358.368,E2 27358.368} C_VEL
LIN {X 0,Y 146.024,Z 683.963,A -85,B 0,C 180,E1 27362.98,E2 27362.98} C_VEL
LIN {X 0,Y 151.703,Z 678.947,A -85,B 0,C 180,E1 27363.57,E2 27363.57} C_VEL
LIN {X 0,Y 153.704,Z 676.973,A -85,B 0,C 180,E1 27364.284,E2 27364.284} C_VEL
LIN {X 0,Y 154.435,Z 675.847,A -85,B 0,C 180,E1 27365.635,E2 27365.635} C_VEL
LIN {X 0,Y 153.983,Z 675.177,A -85,B 0,C 180,E1 27371.35,E2 27371.35} C_VEL
LIN {X 0,Y 151.397,Z 677.504,A -85,B 0,C 180,E1 27376.772,E2 27376.772} C_VEL
LIN {X 0,Y 119.957,Z 701.342,A -85,B 0,C 180,E1 27381.43,E2 27381.43} C_VEL
LIN {X 0,Y 87.079,Z 719.995,A -85,B 0,C 180,E1 27389.616,E2 27389.616} C_VEL
LIN {X 0,Y 55.717,Z 733.338,A -85,B 0,C 180,E1 27407.208,E2 27407.208} C_VEL
LIN {X 0,Y 37.207,Z 740.061,A -85,B 0,C 180,E1 27438.264,E2 27438.264} C_VEL
LIN {X 0,Y 33.463,Z 743.146,A -85,B 0,C 180,E1 27476.907,E2 27476.907} C_VEL
LIN {X 0,Y 53.914,Z 744.15,A -85,B 0,C 180,E1 27523.665,E2 27523.665} C_VEL
LIN {X 0,Y 55.661,Z 746.924,A -85,B 0,C 180,E1 27563.182,E2 27563.182} C_VEL
LIN {X 0,Y 51.715,Z 747.551,A -85,B 0,C 180,E1 27568.551,E2 27568.551} C_VEL
LIN {X 0,Y 35.254,Z 748.725,A -85,B 0,C 180,E1 27604.56,E2 27604.56} C_VEL
LIN {X 0,Y 34.301,Z 748.052,A -85,B 0,C 180,E1 27629.995,E2 27629.995} C_VEL
LIN {X 0,Y 38.654,Z 744.567,A -85,B 0,C 180,E1 27668.487,E2 27668.487} C_VEL
LIN {X 0,Y 50.549,Z 739.746,A -85,B 0,C 180,E1 27690.162,E2 27690.162} C_VEL
LIN {X 0,Y 55.868,Z 737.344,A -85,B 0,C 180,E1 27697.203,E2 27697.203} C_VEL
LIN {X 0,Y 71.141,Z 729.394,A -85,B 0,C 180,E1 27712.815,E2 27712.815} C_VEL
LIN {X 0,Y 72.95,Z 728.556,A -85,B 0,C 180,E1 27713.558,E2 27713.558} C_VEL
LIN {X 0,Y 107.926,Z 710.334,A -85,B 0,C 180,E1 27721.703,E2 27721.703} C_VEL
LIN {X 0,Y 140.644,Z 687.318,A -85,B 0,C 180,E1 27725.696,E2 27725.696} C_VEL
LIN {X 0,Y 148.326,Z 680.835,A -85,B 0,C 180,E1 27726.621,E2 27726.621} C_VEL
LIN {X 0,Y 147.679,Z 680.602,A -85,B 0,C 180,E1 27731.841,E2 27731.841} C_VEL
LIN {X 0,Y 146.698,Z 681.345,A -85,B 0,C 180,E1 27734.176,E2 27734.176} C_VEL
LIN {X 0,Y 113.709,Z 705.017,A -85,B 0,C 180,E1 27738.428,E2 27738.428} C_VEL
LIN {X 0,Y 79.993,Z 722.731,A -85,B 0,C 180,E1 27745.966,E2 27745.966} C_VEL
LIN {X 0,Y 50.228,Z 734.304,A -85,B 0,C 180,E1 27761.099,E2 27761.099} C_VEL
LIN {X 0,Y 29.282,Z 740.938,A -85,B 0,C 180,E1 27795.022,E2 27795.022} C_VEL
LIN {X 0,Y 26.265,Z 743.921,A -85,B 0,C 180,E1 27845.21,E2 27845.21} C_VEL
LIN {X 0,Y 44.977,Z 745.077,A -85,B 0,C 180,E1 27887.871,E2 27887.871} C_VEL
LIN {X 0,Y 46.024,Z 746.98,A -85,B 0,C 180,E1 27919.175,E2 27919.175} C_VEL
LIN {X 0,Y 41.381,Z 747.563,A -85,B 0,C 180,E1 27926.978,E2 27926.978} C_VEL
LIN {X 0,Y 28.202,Z 748.002,A -85,B 0,C 180,E1 27957.522,E2 27957.522} C_VEL
LIN {X 0,Y 26.359,Z 747.299,A -85,B 0,C 180,E1 27989.994,E2 27989.994} C_VEL
LIN {X 0,Y 36.63,Z 742.297,A -85,B 0,C 180,E1 28045.756,E2 28045.756} C_VEL
LIN {X 0,Y 65.243,Z 731.866,A -85,B 0,C 180,E1 28070.498,E2 28070.498} C_VEL
LIN {X 0,Y 72.95,Z 728.556,A -85,B 0,C 180,E1 28073.558,E2 28073.558} C_VEL
LIN {X 0,Y 86.148,Z 721.669,A -85,B 0,C 180,E1 28080.248,E2 28080.248} C_VEL
LIN {X 0,Y 99.9,Z 713.983,A -85,B 0,C 180,E1 28085.081,E2 28085.081} C_VEL
LIN {X 0,Y 133.942,Z 691.825,A -85,B 0,C 180,E1 28088.465,E2 28088.465} C_VEL
LIN {X 0,Y 141.963,Z 685.533,A -85,B 0,C 180,E1 28089.253,E2 28089.253} C_VEL
LIN {X 0,Y 141.707,Z 685.56,A -85,B 0,C 180,E1 28090.728,E2 28090.728} C_VEL
LIN {X 0,Y 137.295,Z 688.933,A -85,B 0,C 180,E1 28091.838,E2 28091.838} C_VEL
LIN {X 0,Y 104.141,Z 710.546,A -85,B 0,C 180,E1 28095.595,E2 28095.595} C_VEL
LIN {X 0,Y 69.731,Z 726.773,A -85,B 0,C 180,E1 28102.662,E2 28102.662} C_VEL
LIN {X 0,Y 38.868,Z 737.165,A -85,B 0,C 180,E1 28118.827,E2 28118.827} C_VEL
LIN {X 0,Y 21.504,Z 741.808,A -85,B 0,C 180,E1 28149.395,E2 28149.395} C_VEL
LIN {X 0,Y 20.001,Z 744.681,A -85,B 0,C 180,E1 28219.215,E2 28219.215} C_VEL
LIN {X 0,Y 31.163,Z 745.57,A -85,B 0,C 180,E1 28246.367,E2 28246.367} C_VEL
LIN {X 0,Y 36.405,Z 745.805,A -85,B 0,C 180,E1 28254.192,E2 28254.192} C_VEL
LIN {X 0,Y 37.03,Z 746.841,A -85,B 0,C 180,E1 28274.446,E2 28274.446} C_VEL
LIN {X 0,Y 32.697,Z 747.236,A -85,B 0,C 180,E1 28282.145,E2 28282.145} C_VEL
LIN {X 0,Y 18.402,Z 746.541,A -85,B 0,C 180,E1 28349.992,E2 28349.992} C_VEL
LIN {X 0,Y 32.75,Z 741.389,A -85,B 0,C 180,E1 28417.604,E2 28417.604} C_VEL
LIN {X 0,Y 66.427,Z 729.923,A -85,B 0,C 180,E1 28438.393,E2 28438.393} C_VEL
LIN {X 0,Y 99.9,Z 713.983,A -85,B 0,C 180,E1 28445.081,E2 28445.081} C_VEL
LIN {X 0,Y 98.699,Z 714.313,A -85,B 0,C 180,E1 28447.057,E2 28447.057} C_VEL
LIN {X 0,Y 93.154,Z 716.825,A -85,B 0,C 180,E1 28449.5,E2 28449.5} C_VEL
LIN {X 0,Y 77.145,Z 723.903,A -85,B 0,C 180,E1 28454.301,E2 28454.301} C_VEL
LIN {X 0,Y 71.545,Z 726.152,A -85,B 0,C 180,E1 28455.594,E2 28455.594} C_VEL
LIN {X 0,Y 34.462,Z 738.111,A -85,B 0,C 180,E1 28468.522,E2 28468.522} C_VEL
LIN {X 0,Y 14.135,Z 742.648,A -85,B 0,C 180,E1 28497.628,E2 28497.628} C_VEL
LIN {X 0,Y 27.167,Z 746.178,A -85,B 0,C 180,E1 28619.951,E2 28619.951} C_VEL
LIN {X 0,Y 28.401,Z 746.451,A -85,B 0,C 180,E1 28626.359,E2 28626.359} C_VEL
LIN {X 0,Y 16.993,Z 746.556,A -85,B 0,C 180,E1 28646.977,E2 28646.977} C_VEL
LIN {X 0,Y 10.427,Z 745.781,A -85,B 0,C 180,E1 28709.985,E2 28709.985} C_VEL
LIN {X 0,Y 30.585,Z 740.476,A -85,B 0,C 180,E1 28791.898,E2 28791.898} C_VEL
LIN {X 0,Y 66.268,Z 728.992,A -85,B 0,C 180,E1 28805.442,E2 28805.442} C_VEL
LIN {X 0,Y 104.262,Z 710.838,A -85,B 0,C 180,E1 28809.989,E2 28809.989} C_VEL
LIN {X 0,Y 107.709,Z 708.83,A -85,B 0,C 180,E1 28810.262,E2 28810.262} C_VEL
LIN {X 0,Y 107.911,Z 708.655,A -85,B 0,C 180,E1 28810.841,E2 28810.841} C_VEL
LIN {X 0,Y 71.545,Z 726.152,A -85,B 0,C 180,E1 28815.594,E2 28815.594} C_VEL
LIN {X 0,Y 58.545,Z 731.082,A -85,B 0,C 180,E1 28815.339,E2 28815.339} C_VEL
LIN {X 0,Y 36.582,Z 738.001,A -85,B 0,C 180,E1 28808.566,E2 28808.566} C_VEL
LIN {X 0,Y 7.6,Z 744.005,A -85,B 0,C 180,E1 28789.815,E2 28789.815} C_VEL
LIN {X 0,Y 2.456,Z 745.011,A -85,B 0,C 180,E1 28709.937,E2 28709.937} C_VEL
LIN {X 0,Y 4.133,Z 745.117,A -85,B 0,C 180,E1 28619.678,E2 28619.678} C_VEL
LIN {X 0,Y 23.85,Z 740.685,A -85,B 0,C 180,E1 28457.792,E2 28457.792} C_VEL
LIN {X 0,Y 46.505,Z 735.072,A -85,B 0,C 180,E1 28452.396,E2 28452.396} C_VEL
LIN {X 0,Y 46.147,Z 735.295,A -85,B 0,C 180,E1 28450.181,E2 28450.181} C_VEL
LIN {X 0,Y 36.582,Z 738.001,A -85,B 0,C 180,E1 28448.566,E2 28448.566} C_VEL
LIN {X 0,Y 35.098,Z 739.936,A -85,B 0,C 180,E1 28448.287,E2 28448.287} C_VEL
LIN {X 0,Y 35.098,Z 786.5,A -85,B 0,C 180,E1 28448.287,E2 28448.287} C_VEL
LIN {X 0,Y 35.098,Z 786.5,A -85,B 0,C 180,E1 28448.287,E2 28448.287}

QRS_NEXT_CUT()
PTP {E1 28616.865,E2 28616.865}
PTP {X 0,Y 607.922,A -85,B 0,C 180,E1 28616.865,E2 28616.865,E3 0,E4 0,E5 0,E6 0}
QRS_SPEED_INIT()
LIN {X 0,Y 607.922,Z 786.5,A -85,B 0,C 180,E1 28616.865,E2 28616.865,E3 0,E4 0,E5 0,E6 0} C_VEL
LIN {X 0,Y 607.922,Z 633.565,A -85,B 0,C 180,E1 28616.865,E2 28616.865} C_VEL
LIN {X 0,Y 607.922,Z 625.003,A -85,B 0,C 180,E1 28616.865,E2 28616.865} C_VEL
LIN {X 0,Y 607.917,Z 623.043,A -85,B 0,C 180,E1 28616.714,E2 28616.714} C_VEL
LIN {X 0,Y 607.913,Z 618.683,A -85,B 0,C 180,E1 28615.093,E2 28615.093} C_VEL
LIN {X 0,Y 607.915,Z 612.881,A -85,B 0,C 180,E1 28613.578,E2 28613.578} C_VEL
LIN {X 0,Y 607.918,Z 605.212,A -85,B 0,C 180,E1 28612.058,E2 28612.058} C_VEL
LIN {X 0,Y 607.919,Z 596.004,A -85,B 0,C 180,E1 28610.629,E2 28610.629} C_VEL
LIN {X 0,Y 607.916,Z 585.33,A -85,B 0,C 180,E1 28609.289,E2 28609.289} C_VEL
LIN {X 0,Y 607.917,Z 572.69,A -85,B 0,C 180,E1 28607.991,E2 28607.991} C_VEL
LIN {X 0,Y 607.918,Z 559.389,A -85,B 0,C 180,E1 28606.881,E2 28606.881} C_VEL
LIN {X 0,Y 607.918,Z 544.347,A -85,B 0,C 180,E1 28605.863,E2 28605.863} C_VEL
LIN {X 0,Y 607.914,Z 529.075,A -85,B 0,C 180,E1 28605.035,E2 28605.035} C_VEL
LIN {X 0,Y 607.897,Z 512.888,A -85,B 0,C 180,E1 28604.351,E2 28604.351} C_VEL
LIN {X 0,Y 607.918,Z 495.905,A -85,B 0,C 180,E1 28603.826,E2 28603.826} C_VEL
LIN {X 0,Y 607.917,Z 478.771,A -85,B 0,C 180,E1 28603.48,E2 28603.48} C_VEL
LIN {X 0,Y 607.914,Z 312.618,A -85,B 0,C 180,E1 28601.442,E2 28601.442} C_VEL
LIN {X 0,Y 607.879,Z 274.291,A -85,B 0,C 180,E1 28598.279,E2 28598.279} C_VEL
LIN {X 0,Y 607.897,Z 237.787,A -85,B 0,C 180,E1 28595.202,E2 28595.202} C_VEL
LIN {X 0,Y 607.9,Z 202.499,A -85,B 0,C 180,E1 28592.152,E2 28592.152} C_VEL
LIN {X 0,Y 607.905,Z 167.877,A -85,B 0,C 180,E1 28589.125,E2 28589.125} C_VEL
LIN {X 0,Y 607.899,Z 166.01,A -85,B 0,C 180,E1 28588.939,E2 28588.939} C_VEL
LIN {X 0,Y 607.889,Z 166.01,A -85,B 0,C 180,E1 28585.827,E2 28585.827} C_VEL
LIN {X 0,Y 607.909,Z 166.015,A -85,B 0,C 180,E1 28582.6,E2 28582.6} C_VEL
LIN {X 0,Y 607.909,Z 166.009,A -85,B 0,C 180,E1 28579.358,E2 28579.358} C_VEL
LIN {X 0,Y 607.916,Z 166.018,A -85,B 0,C 180,E1 28579.19,E2 28579.19} C_VEL
LIN {X 0,Y 607.898,Z 394.901,A -85,B 0,C 180,E1 28576.111,E2 28576.111} C_VEL
LIN {X 0,Y 607.916,Z 462.675,A -85,B 0,C 180,E1 28575.186,E2 28575.186} C_VEL
LIN {X 0,Y 607.913,Z 482.826,A -85,B 0,C 180,E1 28574.745,E2 28574.745} C_VEL
LIN {X 0,Y 607.898,Z 503.655,A -85,B 0,C 180,E1 28574.134,E2 28574.134} C_VEL
LIN {X 0,Y 607.917,Z 523.693,A -85,B 0,C 180,E1 28573.366,E2 28573.366} C_VEL
LIN {X 0,Y 607.917,Z 544.354,A -85,B 0,C 180,E1 28572.397,E2 28572.397} C_VEL
LIN {X 0,Y 607.915,Z 563.421,A -85,B 0,C 180,E1 28571.328,E2 28571.328} C_VEL
LIN {X 0,Y 607.915,Z 582.341,A -85,B 0,C 180,E1 28570.066,E2 28570.066} C_VEL
LIN {X 0,Y 607.91,Z 600.171,A -85,B 0,C 180,E1 28568.683,E2 28568.683} C_VEL
LIN {X 0,Y 607.915,Z 616.885,A -85,B 0,C 180,E1 28567.187,E2 28567.187} C_VEL
LIN {X 0,Y 607.911,Z 632.68,A -85,B 0,C 180,E1 28565.552,E2 28565.552} C_VEL
LIN {X 0,Y 607.916,Z 646.872,A -85,B 0,C 180,E1 28563.84,E2 28563.84} C_VEL
LIN {X 0,Y 607.915,Z 660.152,A -85,B 0,C 180,E1 28561.979,E2 28561.979} C_VEL
LIN {X 0,Y 607.913,Z 671.584,A -85,B 0,C 180,E1 28560.101,E2 28560.101} C_VEL
LIN {X 0,Y 607.908,Z 680.906,A -85,B 0,C 180,E1 28558.274,E2 28558.274} C_VEL
LIN {X 0,Y 607.91,Z 689.355,A -85,B 0,C 180,E1 28556.26,E2 28556.26} C_VEL
LIN {X 0,Y 607.913,Z 695.998,A -85,B 0,C 180,E1 28554.28,E2 28554.28} C_VEL
LIN {X 0,Y 607.915,Z 700.819,A -85,B 0,C 180,E1 28552.33,E2 28552.33} C_VEL
LIN {X 0,Y 607.918,Z 704.393,A -85,B 0,C 180,E1 28550.206,E2 28550.206} C_VEL
LIN {X 0,Y 607.908,Z 706.193,A -85,B 0,C 180,E1 28548.21,E2 28548.21} C_VEL
LIN {X 0,Y 607.916,Z 706.314,A -85,B 0,C 180,E1 28546.139,E2 28546.139} C_VEL
LIN {X 0,Y 607.917,Z 704.735,A -85,B 0,C 180,E1 28543.992,E2 28543.992} C_VEL
LIN {X 0,Y 607.913,Z 701.647,A -85,B 0,C 180,E1 28541.961,E2 28541.961} C_VEL
LIN {X 0,Y 607.911,Z 696.839,A -85,B 0,C 180,E1 28539.945,E2 28539.945} C_VEL
LIN {X 0,Y 607.907,Z 690.084,A -85,B 0,C 180,E1 28537.846,E2 28537.846} C_VEL
LIN {X 0,Y 607.918,Z 682.392,A -85,B 0,C 180,E1 28535.948,E2 28535.948} C_VEL
LIN {X 0,Y 607.916,Z 672.91,A -85,B 0,C 180,E1 28534.056,E2 28534.056} C_VEL
LIN {X 0,Y 607.913,Z 661.092,A -85,B 0,C 180,E1 28532.074,E2 28532.074} C_VEL
LIN {X 0,Y 607.907,Z 648.552,A -85,B 0,C 180,E1 28530.283,E2 28530.283} C_VEL
LIN {X 0,Y 607.913,Z 634.658,A -85,B 0,C 180,E1 28528.586,E2 28528.586} C_VEL
LIN {X 0,Y 607.916,Z 619.51,A -85,B 0,C 180,E1 28526.983,E2 28526.983} C_VEL
LIN {X 0,Y 607.913,Z 601.96,A -85,B 0,C 180,E1 28525.378,E2 28525.378} C_VEL
LIN {X 0,Y 607.918,Z 584.634,A -85,B 0,C 180,E1 28524.005,E2 28524.005} C_VEL
LIN {X 0,Y 607.917,Z 565.678,A -85,B 0,C 180,E1 28522.724,E2 28522.724} C_VEL
LIN {X 0,Y 607.919,Z 546.594,A -85,B 0,C 180,E1 28521.631,E2 28521.631} C_VEL
LIN {X 0,Y 607.909,Z 526.631,A -85,B 0,C 180,E1 28520.665,E2 28520.665} C_VEL
LIN {X 0,Y 607.899,Z 506.767,A -85,B 0,C 180,E1 28519.888,E2 28519.888} C_VEL
LIN {X 0,Y 607.916,Z 484.871,A -85,B 0,C 180,E1 28519.217,E2 28519.217} C_VEL
LIN {X 0,Y 607.912,Z 464.721,A -85,B 0,C 180,E1 28518.761,E2 28518.761} C_VEL
LIN {X 0,Y 607.913,Z 429.39,A -85,B 0,C 180,E1 28518.256,E2 28518.256} C_VEL
LIN {X 0,Y 607.855,Z 220.625,A -85,B 0,C 180,E1 28515.46,E2 28515.46} C_VEL
LIN {X 0,Y 607.891,Z 166.016,A -85,B 0,C 180,E1 28514.718,E2 28514.718} C_VEL
LIN {X 0,Y 607.869,Z 166.014,A -85,B 0,C 180,E1 28511.69,E2 28511.69} C_VEL
LIN {X 0,Y 607.886,Z 166.01,A -85,B 0,C 180,E1 28508.482,E2 28508.482} C_VEL
LIN {X 0,Y 607.903,Z 166.011,A -85,B 0,C 180,E1 28505.41,E2 28505.41} C_VEL
LIN {X 0,Y 607.911,Z 166.013,A -85,B 0,C 180,E1 28502.237,E2 28502.237} C_VEL
LIN {X 0,Y 607.887,Z 166.01,A -85,B 0,C 180,E1 28499.124,E2 28499.124} C_VEL
LIN {X 0,Y 607.855,Z 166.014,A -85,B 0,C 180,E1 28495.995,E2 28495.995} C_VEL
LIN {X 0,Y 607.92,Z 166.014,A -85,B 0,C 180,E1 28492.871,E2 28492.871} C_VEL
LIN {X 0,Y 607.874,Z 166.013,A -85,B 0,C 180,E1 28489.727,E2 28489.727} C_VEL
LIN {X 0,Y 607.895,Z 166.008,A -85,B 0,C 180,E1 28486.436,E2 28486.436} C_VEL
LIN {X 0,Y 607.896,Z 166.011,A -85,B 0,C 180,E1 28483.305,E2 28483.305} C_VEL
LIN {X 0,Y 607.914,Z 166.015,A -85,B 0,C 180,E1 28480.111,E2 28480.111} C_VEL
LIN {X 0,Y 607.896,Z 166.01,A -85,B 0,C 180,E1 28476.895,E2 28476.895} C_VEL
LIN {X 0,Y 607.843,Z 166.015,A -85,B 0,C 180,E1 28473.779,E2 28473.779} C_VEL
LIN {X 0,Y 607.918,Z 166.012,A -85,B 0,C 180,E1 28470.765,E2 28470.765} C_VEL
LIN {X 0,Y 607.885,Z 166.013,A -85,B 0,C 180,E1 28467.635,E2 28467.635} C_VEL
LIN {X 0,Y 607.899,Z 166.008,A -85,B 0,C 180,E1 28464.327,E2 28464.327} C_VEL
LIN {X 0,Y 607.888,Z 166.011,A -85,B 0,C 180,E1 28461.215,E2 28461.215} C_VEL
LIN {X 0,Y 607.907,Z 166.014,A -85,B 0,C 180,E1 28458.012,E2 28458.012} C_VEL
LIN {X 0,Y 607.873,Z 166.013,A -85,B 0,C 180,E1 28454.966,E2 28454.966} C_VEL
LIN {X 0,Y 607.846,Z 166.014,A -85,B 0,C 180,E1 28451.77,E2 28451.77} C_VEL
LIN {X 0,Y 607.915,Z 166.011,A -85,B 0,C 180,E1 28448.703,E2 28448.703} C_VEL
LIN {X 0,Y 607.894,Z 166.013,A -85,B 0,C 180,E1 28445.569,E2 28445.569} C_VEL
LIN {X 0,Y 607.905,Z 166.008,A -85,B 0,C 180,E1 28442.263,E2 28442.263} C_VEL
LIN {X 0,Y 607.881,Z 166.011,A -85,B 0,C 180,E1 28439.152,E2 28439.152} C_VEL
LIN {X 0,Y 607.896,Z 166.014,A -85,B 0,C 180,E1 28435.945,E2 28435.945} C_VEL
LIN {X 0,Y 607.854,Z 166.015,A -85,B 0,C 180,E1 28433.009,E2 28433.009} C_VEL
LIN {X 0,Y 607.859,Z 166.013,A -85,B 0,C 180,E1 28429.768,E2 28429.768} C_VEL
LIN {X 0,Y 607.913,Z 166.011,A -85,B 0,C 180,E1 28426.688,E2 28426.688} C_VEL
LIN {X 0,Y 607.905,Z 166.013,A -85,B 0,C 180,E1 28423.469,E2 28423.469} C_VEL
LIN {X 0,Y 607.909,Z 166.008,A -85,B 0,C 180,E1 28420.186,E2 28420.186} C_VEL
LIN {X 0,Y 607.872,Z 166.012,A -85,B 0,C 180,E1 28417.056,E2 28417.056} C_VEL
LIN {X 0,Y 607.886,Z 166.015,A -85,B 0,C 180,E1 28413.905,E2 28413.905} C_VEL
LIN {X 0,Y 607.857,Z 166.015,A -85,B 0,C 180,E1 28410.972,E2 28410.972} C_VEL
LIN {X 0,Y 607.869,Z 166.012,A -85,B 0,C 180,E1 28407.721,E2 28407.721} C_VEL
LIN {X 0,Y 607.908,Z 166.011,A -85,B 0,C 180,E1 28404.623,E2 28404.623} C_VEL
LIN {X 0,Y 607.908,Z 166.028,A -85,B 0,C 180,E1 28401.423,E2 28401.423} C_VEL
LIN {X 0,Y 607.903,Z 207.966,A -85,B 0,C 180,E1 28398.449,E2 28398.449} C_VEL
LIN {X 0,Y 607.899,Z 248.551,A -85,B 0,C 180,E1 28395.651,E2 28395.651} C_VEL
LIN {X 0,Y 607.88,Z 257.157,A -85,B 0,C 180,E1 28394.881,E2 28394.881} C_VEL
LIN {X 0,Y 607.913,Z 262.496,A -85,B 0,C 180,E1 28394.184,E2 28394.184} C_VEL
LIN {X 0,Y 607.886,Z 264.874,A -85,B 0,C 180,E1 28393.638,E2 28393.638} C_VEL
LIN {X 0,Y 607.901,Z 265.051,A -85,B 0,C 180,E1 28393.228,E2 28393.228} C_VEL
LIN {X 0,Y 607.911,Z 263.843,A -85,B 0,C 180,E1 28392.916,E2 28392.916} C_VEL
LIN {X 0,Y 607.905,Z 261.433,A -85,B 0,C 180,E1 28392.66,E2 28392.66} C_VEL
LIN {X 0,Y 607.909,Z 257.062,A -85,B 0,C 180,E1 28392.435,E2 28392.435} C_VEL
LIN {X 0,Y 607.917,Z 249.247,A -85,B 0,C 180,E1 28392.275,E2 28392.275} C_VEL
LIN {X 0,Y 607.919,Z 243.846,A -85,B 0,C 180,E1 28392.249,E2 28392.249} C_VEL
LIN {X 0,Y 607.918,Z 166.01,A -85,B 0,C 180,E1 28392.231,E2 28392.231} C_VEL
LIN {X 0,Y 607.905,Z 166.016,A -85,B 0,C 180,E1 28388.925,E2 28388.925} C_VEL
LIN {X 0,Y 607.902,Z 166.075,A -85,B 0,C 180,E1 28386.38,E2 28386.38} C_VEL
LIN {X 0,Y 607.918,Z 211.002,A -85,B 0,C 180,E1 28383.382,E2 28383.382} C_VEL
LIN {X 0,Y 607.901,Z 226.81,A -85,B 0,C 180,E1 28382.362,E2 28382.362} C_VEL
LIN {X 0,Y 607.908,Z 444.133,A -85,B 0,C 180,E1 28379.431,E2 28379.431} C_VEL
LIN {X 0,Y 607.915,Z 531.684,A -85,B 0,C 180,E1 28378.247,E2 28378.247} C_VEL
LIN {X 0,Y 607.915,Z 552.224,A -85,B 0,C 180,E1 28377.806,E2 28377.806} C_VEL
LIN {X 0,Y 607.918,Z 572.797,A -85,B 0,C 180,E1 28377.209,E2 28377.209} C_VEL
LIN {X 0,Y 607.914,Z 592.312,A -85,B 0,C 180,E1 28376.47,E2 28376.47} C_VEL
LIN {X 0,Y 607.917,Z 612.761,A -85,B 0,C 180,E1 28375.526,E2 28375.526} C_VEL
LIN {X 0,Y 607.914,Z 632.411,A -85,B 0,C 180,E1 28374.434,E2 28374.434} C_VEL
LIN {X 0,Y 607.918,Z 651,A -85,B 0,C 180,E1 28373.206,E2 28373.206} C_VEL
LIN {X 0,Y 607.91,Z 669.672,A -85,B 0,C 180,E1 28371.77,E2 28371.77} C_VEL
LIN {X 0,Y 607.909,Z 686.643,A -85,B 0,C 180,E1 28370.256,E2 28370.256} C_VEL
LIN {X 0,Y 607.914,Z 702.591,A -85,B 0,C 180,E1 28368.607,E2 28368.607} C_VEL
LIN {X 0,Y 607.916,Z 716.561,A -85,B 0,C 180,E1 28366.925,E2 28366.925} C_VEL
LIN {X 0,Y 607.918,Z 729.903,A -85,B 0,C 180,E1 28365.062,E2 28365.062} C_VEL
LIN {X 0,Y 607.918,Z 741.425,A -85,B 0,C 180,E1 28363.176,E2 28363.176} C_VEL
LIN {X 0,Y 607.903,Z 751.062,A -85,B 0,C 180,E1 28361.287,E2 28361.287} C_VEL
LIN {X 0,Y 607.903,Z 759.464,A -85,B 0,C 180,E1 28359.276,E2 28359.276} C_VEL
LIN {X 0,Y 607.907,Z 766.129,A -85,B 0,C 180,E1 28357.276,E2 28357.276} C_VEL
LIN {X 0,Y 607.912,Z 771.015,A -85,B 0,C 180,E1 28355.285,E2 28355.285} C_VEL
LIN {X 0,Y 607.916,Z 774.447,A -85,B 0,C 180,E1 28353.206,E2 28353.206} C_VEL
LIN {X 0,Y 607.91,Z 776.21,A -85,B 0,C 180,E1 28351.225,E2 28351.225} C_VEL
LIN {X 0,Y 607.902,Z 776.329,A -85,B 0,C 180,E1 28349.246,E2 28349.246} C_VEL
LIN {X 0,Y 607.91,Z 774.896,A -85,B 0,C 180,E1 28347.172,E2 28347.172} C_VEL
LIN {X 0,Y 607.913,Z 771.987,A -85,B 0,C 180,E1 28345.188,E2 28345.188} C_VEL
LIN {X 0,Y 607.916,Z 767.398,A -85,B 0,C 180,E1 28343.199,E2 28343.199} C_VEL
LIN {X 0,Y 607.907,Z 761.237,A -85,B 0,C 180,E1 28341.201,E2 28341.201} C_VEL
LIN {X 0,Y 607.899,Z 753.656,A -85,B 0,C 180,E1 28339.289,E2 28339.289} C_VEL
LIN {X 0,Y 607.9,Z 744.326,A -85,B 0,C 180,E1 28337.364,E2 28337.364} C_VEL
LIN {X 0,Y 607.901,Z 733.744,A -85,B 0,C 180,E1 28335.522,E2 28335.522} C_VEL
LIN {X 0,Y 607.903,Z 721.033,A -85,B 0,C 180,E1 28333.665,E2 28333.665} C_VEL
LIN {X 0,Y 607.914,Z 706.865,A -85,B 0,C 180,E1 28331.889,E2 28331.889} C_VEL
LIN {X 0,Y 607.909,Z 691.099,A -85,B 0,C 180,E1 28330.185,E2 28330.185} C_VEL
LIN {X 0,Y 607.917,Z 674.497,A -85,B 0,C 180,E1 28328.635,E2 28328.635} C_VEL
LIN {X 0,Y 607.915,Z 656.133,A -85,B 0,C 180,E1 28327.16,E2 28327.16} C_VEL
LIN {X 0,Y 607.915,Z 637.682,A -85,B 0,C 180,E1 28325.898,E2 28325.898} C_VEL
LIN {X 0,Y 607.918,Z 617.553,A -85,B 0,C 180,E1 28324.726,E2 28324.726} C_VEL
LIN {X 0,Y 607.912,Z 598.554,A -85,B 0,C 180,E1 28323.793,E2 28323.793} C_VEL
LIN {X 0,Y 607.915,Z 577.963,A -85,B 0,C 180,E1 28322.976,E2 28322.976} C_VEL
LIN {X 0,Y 607.918,Z 556.862,A -85,B 0,C 180,E1 28322.313,E2 28322.313} C_VEL
LIN {X 0,Y 607.918,Z 537.352,A -85,B 0,C 180,E1 28321.86,E2 28321.86} C_VEL
LIN {X 0,Y 607.917,Z 510.286,A -85,B 0,C 180,E1 28321.445,E2 28321.445} C_VEL
LIN {X 0,Y 607.906,Z 284.692,A -85,B 0,C 180,E1 28318.428,E2 28318.428} C_VEL
LIN {X 0,Y 607.908,Z 224.659,A -85,B 0,C 180,E1 28317.603,E2 28317.603} C_VEL
LIN {X 0,Y 607.913,Z 166.015,A -85,B 0,C 180,E1 28314.897,E2 28314.897} C_VEL
LIN {X 0,Y 607.911,Z 166.007,A -85,B 0,C 180,E1 28311.678,E2 28311.678} C_VEL
LIN {X 0,Y 607.883,Z 166.011,A -85,B 0,C 180,E1 28308.451,E2 28308.451} C_VEL
LIN {X 0,Y 607.913,Z 166.077,A -85,B 0,C 180,E1 28307.109,E2 28307.109} C_VEL
LIN {X 0,Y 607.897,Z 167.441,A -85,B 0,C 180,E1 28306.825,E2 28306.825} C_VEL
LIN {X 0,Y 607.881,Z 167.258,A -85,B 0,C 180,E1 28306.499,E2 28306.499} C_VEL
LIN {X 0,Y 607.885,Z 166.011,A -85,B 0,C 180,E1 28306.174,E2 28306.174} C_VEL
LIN {X 0,Y 607.898,Z 166.014,A -85,B 0,C 180,E1 28302.917,E2 28302.917} C_VEL
LIN {X 0,Y 607.913,Z 166.006,A -85,B 0,C 180,E1 28299.777,E2 28299.777} C_VEL
LIN {X 0,Y 607.871,Z 166.012,A -85,B 0,C 180,E1 28296.612,E2 28296.612} C_VEL
LIN {X 0,Y 607.916,Z 166.012,A -85,B 0,C 180,E1 28293.434,E2 28293.434} C_VEL
LIN {X 0,Y 607.861,Z 166.193,A -85,B 0,C 180,E1 28290.574,E2 28290.574} C_VEL
LIN {X 0,Y 607.89,Z 184.359,A -85,B 0,C 180,E1 28289.08,E2 28289.08} C_VEL
LIN {X 0,Y 607.911,Z 219.843,A -85,B 0,C 180,E1 28286.049,E2 28286.049} C_VEL
LIN {X 0,Y 607.903,Z 257.514,A -85,B 0,C 180,E1 28282.916,E2 28282.916} C_VEL
LIN {X 0,Y 607.896,Z 295.798,A -85,B 0,C 180,E1 28279.805,E2 28279.805} C_VEL
LIN {X 0,Y 607.855,Z 312.633,A -85,B 0,C 180,E1 28278.46,E2 28278.46} C_VEL
LIN {X 0,Y 607.881,Z 481.775,A -85,B 0,C 180,E1 28276.385,E2 28276.385} C_VEL
LIN {X 0,Y 607.912,Z 499.29,A -85,B 0,C 180,E1 28275.991,E2 28275.991} C_VEL
LIN {X 0,Y 607.915,Z 515.663,A -85,B 0,C 180,E1 28275.453,E2 28275.453} C_VEL
LIN {X 0,Y 607.915,Z 531.915,A -85,B 0,C 180,E1 28274.736,E2 28274.736} C_VEL
LIN {X 0,Y 607.919,Z 546.884,A -85,B 0,C 180,E1 28273.894,E2 28273.894} C_VEL
LIN {X 0,Y 607.918,Z 561.376,A -85,B 0,C 180,E1 28272.877,E2 28272.877} C_VEL
LIN {X 0,Y 607.917,Z 574.784,A -85,B 0,C 180,E1 28271.719,E2 28271.719} C_VEL
LIN {X 0,Y 607.915,Z 587.243,A -85,B 0,C 180,E1 28270.405,E2 28270.405} C_VEL
LIN {X 0,Y 607.913,Z 597.407,A -85,B 0,C 180,E1 28269.084,E2 28269.084} C_VEL
LIN {X 0,Y 607.915,Z 606.283,A -85,B 0,C 180,E1 28267.656,E2 28267.656} C_VEL
LIN {X 0,Y 607.915,Z 613.714,A -85,B 0,C 180,E1 28266.137,E2 28266.137} C_VEL
LIN {X 0,Y 607.917,Z 619.604,A -85,B 0,C 180,E1 28264.528,E2 28264.528} C_VEL
LIN {X 0,Y 607.914,Z 623.635,A -85,B 0,C 180,E1 28262.922,E2 28262.922} C_VEL
LIN {X 0,Y 607.913,Z 625.885,A -85,B 0,C 180,E1 28261.319,E2 28261.319} C_VEL
LIN {X 0,Y 607.913,Z 626.429,A -85,B 0,C 180,E1 28259.623,E2 28259.623} C_VEL
LIN {X 0,Y 607.912,Z 625.143,A -85,B 0,C 180,E1 28257.926,E2 28257.926} C_VEL
LIN {X 0,Y 607.917,Z 623.043,A -85,B 0,C 180,E1 28256.714,E2 28256.714} C_VEL
LIN {X 0,Y 606.916,Z 621.383,A -85,B 0,C 180,E1 28256.005,E2 28256.005} C_VEL
LIN {X 0,Y 602.462,Z 617.677,A -85,B 0,C 180,E1 28254.74,E2 28254.74} C_VEL
LIN {X 0,Y 600.124,Z 614.429,A -85,B 0,C 180,E1 28253.859,E2 28253.859} C_VEL
LIN {X 0,Y 599.922,Z 613.175,A -85,B 0,C 180,E1 28253.562,E2 28253.562} C_VEL
LIN {X 0,Y 599.934,Z 605.735,A -85,B 0,C 180,E1 28252.048,E2 28252.048} C_VEL
LIN {X 0,Y 599.953,Z 596.702,A -85,B 0,C 180,E1 28250.6,E2 28250.6} C_VEL
LIN {X 0,Y 599.974,Z 586.176,A -85,B 0,C 180,E1 28249.242,E2 28249.242} C_VEL
LIN {X 0,Y 600.006,Z 573.7,A -85,B 0,C 180,E1 28247.928,E2 28247.928} C_VEL
LIN {X 0,Y 600.051,Z 560.04,A -85,B 0,C 180,E1 28246.755,E2 28246.755} C_VEL
LIN {X 0,Y 600.093,Z 545.148,A -85,B 0,C 180,E1 28245.724,E2 28245.724} C_VEL
LIN {X 0,Y 600.134,Z 529.071,A -85,B 0,C 180,E1 28244.836,E2 28244.836} C_VEL
LIN {X 0,Y 600.159,Z 512.884,A -85,B 0,C 180,E1 28244.144,E2 28244.144} C_VEL
LIN {X 0,Y 600.22,Z 495.577,A -85,B 0,C 180,E1 28243.606,E2 28243.606} C_VEL
LIN {X 0,Y 600.245,Z 478.093,A -85,B 0,C 180,E1 28243.252,E2 28243.252} C_VEL
LIN {X 0,Y 600.161,Z 312.611,A -85,B 0,C 180,E1 28241.193,E2 28241.193} C_VEL
LIN {X 0,Y 600.213,Z 275.5,A -85,B 0,C 180,E1 28238.09,E2 28238.09} C_VEL
LIN {X 0,Y 600.33,Z 239.605,A -85,B 0,C 180,E1 28235.026,E2 28235.026} C_VEL
LIN {X 0,Y 600.44,Z 204.491,A -85,B 0,C 180,E1 28231.953,E2 28231.953} C_VEL
LIN {X 0,Y 600.35,Z 173.973,A -85,B 0,C 180,E1 28229.305,E2 28229.305} C_VEL
LIN {X 0,Y 600.146,Z 167.99,A -85,B 0,C 180,E1 28228.792,E2 28228.792} C_VEL
LIN {X 0,Y 599.962,Z 167.004,A -85,B 0,C 180,E1 28228.67,E2 28228.67} C_VEL
LIN {X 0,Y 599.97,Z 166.996,A -85,B 0,C 180,E1 28225.413,E2 28225.413} C_VEL
LIN {X 0,Y 599.94,Z 167.002,A -85,B 0,C 180,E1 28222.17,E2 28222.17} C_VEL
LIN {X 0,Y 599.961,Z 167.144,A -85,B 0,C 180,E1 28219.655,E2 28219.655} C_VEL
LIN {X 0,Y 601.14,Z 170.975,A -85,B 0,C 180,E1 28219.53,E2 28219.53} C_VEL
LIN {X 0,Y 600.905,Z 398.323,A -85,B 0,C 180,E1 28216.437,E2 28216.437} C_VEL
LIN {X 0,Y 600.859,Z 463.167,A -85,B 0,C 180,E1 28215.54,E2 28215.54} C_VEL
LIN {X 0,Y 600.793,Z 483.923,A -85,B 0,C 180,E1 28215.075,E2 28215.075} C_VEL
LIN {X 0,Y 600.695,Z 505.182,A -85,B 0,C 180,E1 28214.432,E2 28214.432} C_VEL
LIN {X 0,Y 600.642,Z 525.169,A -85,B 0,C 180,E1 28213.65,E2 28213.65} C_VEL
LIN {X 0,Y 600.537,Z 545.738,A -85,B 0,C 180,E1 28212.659,E2 28212.659} C_VEL
LIN {X 0,Y 600.442,Z 564.56,A -85,B 0,C 180,E1 28211.58,E2 28211.58} C_VEL
LIN {X 0,Y 600.349,Z 584.01,A -85,B 0,C 180,E1 28210.256,E2 28210.256} C_VEL
LIN {X 0,Y 600.246,Z 601.02,A -85,B 0,C 180,E1 28208.902,E2 28208.902} C_VEL
LIN {X 0,Y 600.163,Z 618.17,A -85,B 0,C 180,E1 28207.331,E2 28207.331} C_VEL
LIN {X 0,Y 600.09,Z 633.801,A -85,B 0,C 180,E1 28205.674,E2 28205.674} C_VEL
LIN {X 0,Y 600.044,Z 648.034,A -85,B 0,C 180,E1 28203.919,E2 28203.919} C_VEL
LIN {X 0,Y 599.998,Z 660.599,A -85,B 0,C 180,E1 28202.113,E2 28202.113} C_VEL
LIN {X 0,Y 599.959,Z 671.906,A -85,B 0,C 180,E1 28200.219,E2 28200.219} C_VEL
LIN {X 0,Y 599.939,Z 681.749,A -85,B 0,C 180,E1 28198.25,E2 28198.25} C_VEL
LIN {X 0,Y 599.922,Z 689.751,A -85,B 0,C 180,E1 28196.277,E2 28196.277} C_VEL
LIN {X 0,Y 599.92,Z 696.455,A -85,B 0,C 180,E1 28194.205,E2 28194.205} C_VEL
LIN {X 0,Y 599.918,Z 701.189,A -85,B 0,C 180,E1 28192.231,E2 28192.231} C_VEL
LIN {X 0,Y 599.917,Z 704.475,A -85,B 0,C 180,E1 28190.182,E2 28190.182} C_VEL
LIN {X 0,Y 599.912,Z 706.222,A -85,B 0,C 180,E1 28188.16,E2 28188.16} C_VEL
LIN {X 0,Y 599.915,Z 706.322,A -85,B 0,C 180,E1 28186.161,E2 28186.161} C_VEL
LIN {X 0,Y 599.917,Z 704.776,A -85,B 0,C 180,E1 28183.985,E2 28183.985} C_VEL
LIN {X 0,Y 599.913,Z 701.713,A -85,B 0,C 180,E1 28181.927,E2 28181.927} C_VEL
LIN {X 0,Y 599.912,Z 696.93,A -85,B 0,C 180,E1 28179.885,E2 28179.885} C_VEL
LIN {X 0,Y 599.915,Z 690.212,A -85,B 0,C 180,E1 28177.759,E2 28177.759} C_VEL
LIN {X 0,Y 599.943,Z 682.542,A -85,B 0,C 180,E1 28175.835,E2 28175.835} C_VEL
LIN {X 0,Y 599.963,Z 673.107,A -85,B 0,C 180,E1 28173.918,E2 28173.918} C_VEL
LIN {X 0,Y 599.996,Z 661.336,A -85,B 0,C 180,E1 28171.91,E2 28171.91} C_VEL
LIN {X 0,Y 600.04,Z 648.847,A -85,B 0,C 180,E1 28170.096,E2 28170.096} C_VEL
LIN {X 0,Y 600.093,Z 634.181,A -85,B 0,C 180,E1 28168.282,E2 28168.282} C_VEL
LIN {X 0,Y 600.159,Z 618.952,A -85,B 0,C 180,E1 28166.657,E2 28166.657} C_VEL
LIN {X 0,Y 600.245,Z 601.854,A -85,B 0,C 180,E1 28165.079,E2 28165.079} C_VEL
LIN {X 0,Y 600.352,Z 584.504,A -85,B 0,C 180,E1 28163.689,E2 28163.689} C_VEL
LIN {X 0,Y 600.44,Z 564.794,A -85,B 0,C 180,E1 28162.345,E2 28162.345} C_VEL
LIN {X 0,Y 600.54,Z 545.485,A -85,B 0,C 180,E1 28161.237,E2 28161.237} C_VEL
LIN {X 0,Y 600.637,Z 524.308,A -85,B 0,C 180,E1 28160.224,E2 28160.224} C_VEL
LIN {X 0,Y 600.697,Z 504.409,A -85,B 0,C 180,E1 28159.45,E2 28159.45} C_VEL
LIN {X 0,Y 600.799,Z 483.152,A -85,B 0,C 180,E1 28158.815,E2 28158.815} C_VEL
LIN {X 0,Y 600.854,Z 461.985,A -85,B 0,C 180,E1 28158.351,E2 28158.351} C_VEL
LIN {X 0,Y 600.986,Z 330.332,A -85,B 0,C 180,E1 28156.559,E2 28156.559} C_VEL
LIN {X 0,Y 600.958,Z 170.07,A -85,B 0,C 180,E1 28154.357,E2 28154.357} C_VEL
LIN {X 0,Y 599.909,Z 167.006,A -85,B 0,C 180,E1 28154.236,E2 28154.236} C_VEL
LIN {X 0,Y 599.976,Z 167.004,A -85,B 0,C 180,E1 28151.187,E2 28151.187} C_VEL
LIN {X 0,Y 599.947,Z 167.002,A -85,B 0,C 180,E1 28147.977,E2 28147.977} C_VEL
LIN {X 0,Y 599.972,Z 166.996,A -85,B 0,C 180,E1 28144.746,E2 28144.746} C_VEL
LIN {X 0,Y 599.946,Z 167,A -85,B 0,C 180,E1 28141.534,E2 28141.534} C_VEL
LIN {X 0,Y 599.969,Z 167.003,A -85,B 0,C 180,E1 28138.335,E2 28138.335} C_VEL
LIN {X 0,Y 599.926,Z 167.003,A -85,B 0,C 180,E1 28135.251,E2 28135.251} C_VEL
LIN {X 0,Y 599.915,Z 167.002,A -85,B 0,C 180,E1 28132.031,E2 28132.031} C_VEL
LIN {X 0,Y 599.977,Z 166.998,A -85,B 0,C 180,E1 28128.959,E2 28128.959} C_VEL
LIN {X 0,Y 599.97,Z 167.003,A -85,B 0,C 180,E1 28125.712,E2 28125.712} C_VEL
LIN {X 0,Y 599.967,Z 166.998,A -85,B 0,C 180,E1 28122.416,E2 28122.416} C_VEL
LIN {X 0,Y 599.938,Z 167,A -85,B 0,C 180,E1 28119.295,E2 28119.295} C_VEL
LIN {X 0,Y 599.935,Z 167.003,A -85,B 0,C 180,E1 28116.069,E2 28116.069} C_VEL
LIN {X 0,Y 599.943,Z 167.004,A -85,B 0,C 180,E1 28113.023,E2 28113.023} C_VEL
LIN {X 0,Y 599.924,Z 167.002,A -85,B 0,C 180,E1 28109.89,E2 28109.89} C_VEL
LIN {X 0,Y 599.976,Z 166.996,A -85,B 0,C 180,E1 28106.716,E2 28106.716} C_VEL
LIN {X 0,Y 599.971,Z 167.001,A -85,B 0,C 180,E1 28103.472,E2 28103.472} C_VEL
LIN {X 0,Y 599.972,Z 167,A -85,B 0,C 180,E1 28100.241,E2 28100.241} C_VEL
LIN {X 0,Y 599.931,Z 167,A -85,B 0,C 180,E1 28097.157,E2 28097.157} C_VEL
LIN {X 0,Y 599.915,Z 167.003,A -85,B 0,C 180,E1 28093.887,E2 28093.887} C_VEL
LIN {X 0,Y 599.974,Z 167.004,A -85,B 0,C 180,E1 28090.758,E2 28090.758} C_VEL
LIN {X 0,Y 599.938,Z 167.001,A -85,B 0,C 180,E1 28087.566,E2 28087.566} C_VEL
LIN {X 0,Y 599.963,Z 166.995,A -85,B 0,C 180,E1 28084.301,E2 28084.301} C_VEL
LIN {X 0,Y 599.953,Z 167,A -85,B 0,C 180,E1 28081.146,E2 28081.146} C_VEL
LIN {X 0,Y 599.969,Z 167.004,A -85,B 0,C 180,E1 28077.899,E2 28077.899} C_VEL
LIN {X 0,Y 599.947,Z 167,A -85,B 0,C 180,E1 28074.741,E2 28074.741} C_VEL
LIN {X 0,Y 599.903,Z 167.003,A -85,B 0,C 180,E1 28071.566,E2 28071.566} C_VEL
LIN {X 0,Y 599.974,Z 166.998,A -85,B 0,C 180,E1 28068.464,E2 28068.464} C_VEL
LIN {X 0,Y 599.97,Z 167.003,A -85,B 0,C 180,E1 28065.228,E2 28065.228} C_VEL
LIN {X 0,Y 599.961,Z 166.999,A -85,B 0,C 180,E1 28061.942,E2 28061.942} C_VEL
LIN {X 0,Y 599.949,Z 166.998,A -85,B 0,C 180,E1 28058.799,E2 28058.799} C_VEL
LIN {X 0,Y 599.931,Z 167.003,A -85,B 0,C 180,E1 28055.482,E2 28055.482} C_VEL
LIN {X 0,Y 599.97,Z 167.003,A -85,B 0,C 180,E1 28052.401,E2 28052.401} C_VEL
LIN {X 0,Y 599.917,Z 167.004,A -85,B 0,C 180,E1 28049.316,E2 28049.316} C_VEL
LIN {X 0,Y 599.958,Z 166.999,A -85,B 0,C 180,E1 28046.093,E2 28046.093} C_VEL
LIN {X 0,Y 599.968,Z 167.004,A -85,B 0,C 180,E1 28042.895,E2 28042.895} C_VEL
LIN {X 0,Y 599.987,Z 167.172,A -85,B 0,C 180,E1 28042.021,E2 28042.021} C_VEL
LIN {X 0,Y 601.399,Z 171.022,A -85,B 0,C 180,E1 28041.614,E2 28041.614} C_VEL
LIN {X 0,Y 601.209,Z 213.252,A -85,B 0,C 180,E1 28038.595,E2 28038.595} C_VEL
LIN {X 0,Y 601.483,Z 256.619,A -85,B 0,C 180,E1 28035.586,E2 28035.586} C_VEL
LIN {X 0,Y 602.457,Z 264.211,A -85,B 0,C 180,E1 28034.941,E2 28034.941} C_VEL
LIN {X 0,Y 603.485,Z 269.414,A -85,B 0,C 180,E1 28034.296,E2 28034.296} C_VEL
LIN {X 0,Y 604.365,Z 272.064,A -85,B 0,C 180,E1 28033.7,E2 28033.7} C_VEL
LIN {X 0,Y 604.967,Z 272.483,A -85,B 0,C 180,E1 28033.176,E2 28033.176} C_VEL
LIN {X 0,Y 605.179,Z 271.427,A -85,B 0,C 180,E1 28032.769,E2 28032.769} C_VEL
LIN {X 0,Y 605.003,Z 268.718,A -85,B 0,C 180,E1 28032.352,E2 28032.352} C_VEL
LIN {X 0,Y 604.415,Z 264.274,A -85,B 0,C 180,E1 28032.017,E2 28032.017} C_VEL
LIN {X 0,Y 603.525,Z 257.946,A -85,B 0,C 180,E1 28031.795,E2 28031.795} C_VEL
LIN {X 0,Y 602.65,Z 248.12,A -85,B 0,C 180,E1 28031.694,E2 28031.694} C_VEL
LIN {X 0,Y 602.541,Z 171.939,A -85,B 0,C 180,E1 28031.683,E2 28031.683} C_VEL
LIN {X 0,Y 600.55,Z 169.174,A -85,B 0,C 180,E1 28031.469,E2 28031.469} C_VEL
LIN {X 0,Y 599.954,Z 167.005,A -85,B 0,C 180,E1 28031.389,E2 28031.389} C_VEL
LIN {X 0,Y 599.973,Z 167,A -85,B 0,C 180,E1 28028.069,E2 28028.069} C_VEL
LIN {X 0,Y 599.967,Z 167.151,A -85,B 0,C 180,E1 28026.866,E2 28026.866} C_VEL
LIN {X 0,Y 601.044,Z 170.821,A -85,B 0,C 180,E1 28026.536,E2 28026.536} C_VEL
LIN {X 0,Y 600.869,Z 215.564,A -85,B 0,C 180,E1 28023.522,E2 28023.522} C_VEL
LIN {X 0,Y 600.927,Z 227.209,A -85,B 0,C 180,E1 28022.779,E2 28022.779} C_VEL
LIN {X 0,Y 601.047,Z 303.036,A -85,B 0,C 180,E1 28021.722,E2 28021.722} C_VEL
LIN {X 0,Y 600.859,Z 532.042,A -85,B 0,C 180,E1 28018.604,E2 28018.604} C_VEL
LIN {X 0,Y 600.796,Z 553.413,A -85,B 0,C 180,E1 28018.134,E2 28018.134} C_VEL
LIN {X 0,Y 600.72,Z 574.316,A -85,B 0,C 180,E1 28017.508,E2 28017.508} C_VEL
LIN {X 0,Y 600.641,Z 594.87,A -85,B 0,C 180,E1 28016.709,E2 28016.709} C_VEL
LIN {X 0,Y 600.54,Z 614.94,A -85,B 0,C 180,E1 28015.747,E2 28015.747} C_VEL
LIN {X 0,Y 600.446,Z 634.124,A -85,B 0,C 180,E1 28014.653,E2 28014.653} C_VEL
LIN {X 0,Y 600.355,Z 653.292,A -85,B 0,C 180,E1 28013.352,E2 28013.352} C_VEL
LIN {X 0,Y 600.248,Z 670.885,A -85,B 0,C 180,E1 28011.96,E2 28011.96} C_VEL
LIN {X 0,Y 600.157,Z 688.166,A -85,B 0,C 180,E1 28010.377,E2 28010.377} C_VEL
LIN {X 0,Y 600.098,Z 703.47,A -85,B 0,C 180,E1 28008.758,E2 28008.758} C_VEL
LIN {X 0,Y 600.044,Z 718.118,A -85,B 0,C 180,E1 28006.954,E2 28006.954} C_VEL
LIN {X 0,Y 599.995,Z 730.547,A -85,B 0,C 180,E1 28005.167,E2 28005.167} C_VEL
LIN {X 0,Y 599.962,Z 742.253,A -85,B 0,C 180,E1 28003.198,E2 28003.198} C_VEL
LIN {X 0,Y 599.934,Z 751.988,A -85,B 0,C 180,E1 28001.244,E2 28001.244} C_VEL
LIN {X 0,Y 599.915,Z 759.822,A -85,B 0,C 180,E1 27999.304,E2 27999.304} C_VEL
LIN {X 0,Y 599.911,Z 766.386,A -85,B 0,C 180,E1 27997.277,E2 27997.277} C_VEL
LIN {X 0,Y 599.914,Z 771.018,A -85,B 0,C 180,E1 27995.355,E2 27995.355} C_VEL
LIN {X 0,Y 599.917,Z 774.45,A -85,B 0,C 180,E1 27993.248,E2 27993.248} C_VEL
LIN {X 0,Y 599.916,Z 776.243,A -85,B 0,C 180,E1 27991.146,E2 27991.146} C_VEL
LIN {X 0,Y 599.908,Z 776.31,A -85,B 0,C 180,E1 27989.14,E2 27989.14} C_VEL
LIN {X 0,Y 599.915,Z 774.786,A -85,B 0,C 180,E1 27987.038,E2 27987.038} C_VEL
LIN {X 0,Y 599.918,Z 771.634,A -85,B 0,C 180,E1 27984.932,E2 27984.932} C_VEL
LIN {X 0,Y 599.92,Z 766.894,A -85,B 0,C 180,E1 27982.915,E2 27982.915} C_VEL
LIN {X 0,Y 599.92,Z 760.176,A -85,B 0,C 180,E1 27980.793,E2 27980.793} C_VEL
LIN {X 0,Y 599.939,Z 752.429,A -85,B 0,C 180,E1 27978.853,E2 27978.853} C_VEL
LIN {X 0,Y 599.958,Z 742.771,A -85,B 0,C 180,E1 27976.9,E2 27976.9} C_VEL
LIN {X 0,Y 599.993,Z 731.187,A -85,B 0,C 180,E1 27974.932,E2 27974.932} C_VEL
LIN {X 0,Y 600.038,Z 718.884,A -85,B 0,C 180,E1 27973.145,E2 27973.145} C_VEL
LIN {X 0,Y 600.092,Z 704.317,A -85,B 0,C 180,E1 27971.343,E2 27971.343} C_VEL
LIN {X 0,Y 600.159,Z 689.027,A -85,B 0,C 180,E1 27969.71,E2 27969.71} C_VEL
LIN {X 0,Y 600.246,Z 671.484,A -85,B 0,C 180,E1 27968.091,E2 27968.091} C_VEL
LIN {X 0,Y 600.352,Z 654.015,A -85,B 0,C 180,E1 27966.7,E2 27966.7} C_VEL
LIN {X 0,Y 600.435,Z 634.893,A -85,B 0,C 180,E1 27965.396,E2 27965.396} C_VEL
LIN {X 0,Y 600.538,Z 615.743,A -85,B 0,C 180,E1 27964.296,E2 27964.296} C_VEL
LIN {X 0,Y 600.634,Z 595.562,A -85,B 0,C 180,E1 27963.32,E2 27963.32} C_VEL
LIN {X 0,Y 600.715,Z 575.014,A -85,B 0,C 180,E1 27962.517,E2 27962.517} C_VEL
LIN {X 0,Y 600.796,Z 553.582,A -85,B 0,C 180,E1 27961.87,E2 27961.87} C_VEL
LIN {X 0,Y 600.86,Z 532.234,A -85,B 0,C 180,E1 27961.399,E2 27961.399} C_VEL
LIN {X 0,Y 600.989,Z 394.114,A -85,B 0,C 180,E1 27959.52,E2 27959.52} C_VEL
LIN {X 0,Y 600.996,Z 224.994,A -85,B 0,C 180,E1 27957.194,E2 27957.194} C_VEL
LIN {X 0,Y 601.102,Z 170.237,A -85,B 0,C 180,E1 27954.644,E2 27954.644} C_VEL
LIN {X 0,Y 599.951,Z 167.001,A -85,B 0,C 180,E1 27954.381,E2 27954.381} C_VEL
LIN {X 0,Y 599.97,Z 167.003,A -85,B 0,C 180,E1 27951.199,E2 27951.199} C_VEL
LIN {X 0,Y 599.964,Z 167.122,A -85,B 0,C 180,E1 27948.594,E2 27948.594} C_VEL
LIN {X 0,Y 600.93,Z 169.968,A -85,B 0,C 180,E1 27948.482,E2 27948.482} C_VEL
LIN {X 0,Y 602.737,Z 172.132,A -85,B 0,C 180,E1 27948.206,E2 27948.206} C_VEL
LIN {X 0,Y 604.855,Z 173.398,A -85,B 0,C 180,E1 27947.717,E2 27947.717} C_VEL
LIN {X 0,Y 605.824,Z 173.898,A -85,B 0,C 180,E1 27947.287,E2 27947.287} C_VEL
LIN {X 0,Y 605.751,Z 175.186,A -85,B 0,C 180,E1 27946.85,E2 27946.85} C_VEL
LIN {X 0,Y 605.383,Z 174.95,A -85,B 0,C 180,E1 27946.471,E2 27946.471} C_VEL
LIN {X 0,Y 604.595,Z 173.297,A -85,B 0,C 180,E1 27946.004,E2 27946.004} C_VEL
LIN {X 0,Y 602.57,Z 171.968,A -85,B 0,C 180,E1 27945.521,E2 27945.521} C_VEL
LIN {X 0,Y 600.762,Z 169.6,A -85,B 0,C 180,E1 27945.153,E2 27945.153} C_VEL
LIN {X 0,Y 599.962,Z 167.005,A -85,B 0,C 180,E1 27944.905,E2 27944.905} C_VEL
LIN {X 0,Y 599.977,Z 166.997,A -85,B 0,C 180,E1 27941.677,E2 27941.677} C_VEL
LIN {X 0,Y 599.934,Z 167,A -85,B 0,C 180,E1 27938.558,E2 27938.558} C_VEL
LIN {X 0,Y 599.976,Z 167.001,A -85,B 0,C 180,E1 27935.42,E2 27935.42} C_VEL
LIN {X 0,Y 599.926,Z 167.001,A -85,B 0,C 180,E1 27932.329,E2 27932.329} C_VEL
LIN {X 0,Y 599.954,Z 167.204,A -85,B 0,C 180,E1 27930.698,E2 27930.698} C_VEL
LIN {X 0,Y 600.307,Z 187.98,A -85,B 0,C 180,E1 27929.101,E2 27929.101} C_VEL
LIN {X 0,Y 600.403,Z 207.927,A -85,B 0,C 180,E1 27927.425,E2 27927.425} C_VEL
LIN {X 0,Y 600.339,Z 243.509,A -85,B 0,C 180,E1 27924.396,E2 27924.396} C_VEL
LIN {X 0,Y 600.237,Z 282.109,A -85,B 0,C 180,E1 27921.19,E2 27921.19} C_VEL
LIN {X 0,Y 600.168,Z 313.026,A -85,B 0,C 180,E1 27918.701,E2 27918.701} C_VEL
LIN {X 0,Y 600.2,Z 482.306,A -85,B 0,C 180,E1 27916.591,E2 27916.591} C_VEL
LIN {X 0,Y 600.203,Z 500.178,A -85,B 0,C 180,E1 27916.177,E2 27916.177} C_VEL
LIN {X 0,Y 600.169,Z 516.841,A -85,B 0,C 180,E1 27915.613,E2 27915.613} C_VEL
LIN {X 0,Y 600.127,Z 533.225,A -85,B 0,C 180,E1 27914.867,E2 27914.867} C_VEL
LIN {X 0,Y 600.082,Z 548.42,A -85,B 0,C 180,E1 27913.981,E2 27913.981} C_VEL
LIN {X 0,Y 600.038,Z 562.594,A -85,B 0,C 180,E1 27912.951,E2 27912.951} C_VEL
LIN {X 0,Y 600.002,Z 576.311,A -85,B 0,C 180,E1 27911.73,E2 27911.73} C_VEL
LIN {X 0,Y 599.968,Z 587.907,A -85,B 0,C 180,E1 27910.466,E2 27910.466} C_VEL
LIN {X 0,Y 599.943,Z 598.052,A -85,B 0,C 180,E1 27909.109,E2 27909.109} C_VEL
LIN {X 0,Y 599.932,Z 607.323,A -85,B 0,C 180,E1 27907.565,E2 27907.565} C_VEL
LIN {X 0,Y 599.921,Z 614.529,A -85,B 0,C 180,E1 27906.027,E2 27906.027} C_VEL
LIN {X 0,Y 599.919,Z 620.198,A -85,B 0,C 180,E1 27904.397,E2 27904.397} C_VEL
LIN {X 0,Y 599.913,Z 623.976,A -85,B 0,C 180,E1 27902.77,E2 27902.77} C_VEL
LIN {X 0,Y 599.912,Z 626.088,A -85,B 0,C 180,E1 27901.05,E2 27901.05} C_VEL
LIN {X 0,Y 599.916,Z 626.364,A -85,B 0,C 180,E1 27899.331,E2 27899.331} C_VEL
LIN {X 0,Y 599.909,Z 624.902,A -85,B 0,C 180,E1 27897.707,E2 27897.707} C_VEL
LIN {X 0,Y 599.914,Z 621.704,A -85,B 0,C 180,E1 27896.081,E2 27896.081} C_VEL
LIN {X 0,Y 599.921,Z 616.708,A -85,B 0,C 180,E1 27894.452,E2 27894.452} C_VEL
LIN {X 0,Y 599.922,Z 613.175,A -85,B 0,C 180,E1 27893.562,E2 27893.562} C_VEL
LIN {X 0,Y 598.925,Z 610.179,A -85,B 0,C 180,E1 27892.884,E2 27892.884} C_VEL
LIN {X 0,Y 594.134,Z 603.617,A -85,B 0,C 180,E1 27891.595,E2 27891.595} C_VEL
LIN {X 0,Y 592.167,Z 599.274,A -85,B 0,C 180,E1 27890.865,E2 27890.865} C_VEL
LIN {X 0,Y 591.983,Z 597.495,A -85,B 0,C 180,E1 27890.591,E2 27890.591} C_VEL
LIN {X 0,Y 592.032,Z 587.013,A -85,B 0,C 180,E1 27889.195,E2 27889.195} C_VEL
LIN {X 0,Y 592.095,Z 574.994,A -85,B 0,C 180,E1 27887.891,E2 27887.891} C_VEL
LIN {X 0,Y 592.176,Z 561.268,A -85,B 0,C 180,E1 27886.675,E2 27886.675} C_VEL
LIN {X 0,Y 592.268,Z 546.731,A -85,B 0,C 180,E1 27885.631,E2 27885.631} C_VEL
LIN {X 0,Y 592.353,Z 531.057,A -85,B 0,C 180,E1 27884.733,E2 27884.733} C_VEL
LIN {X 0,Y 592.422,Z 514.348,A -85,B 0,C 180,E1 27883.989,E2 27883.989} C_VEL
LIN {X 0,Y 592.517,Z 497.32,A -85,B 0,C 180,E1 27883.434,E2 27883.434} C_VEL
LIN {X 0,Y 592.576,Z 479.778,A -85,B 0,C 180,E1 27883.055,E2 27883.055} C_VEL
LIN {X 0,Y 592.525,Z 313.497,A -85,B 0,C 180,E1 27880.964,E2 27880.964} C_VEL
LIN {X 0,Y 592.416,Z 311.994,A -85,B 0,C 180,E1 27880.887,E2 27880.887} C_VEL
LIN {X 0,Y 592.563,Z 274.884,A -85,B 0,C 180,E1 27877.74,E2 27877.74} C_VEL
LIN {X 0,Y 592.761,Z 238.38,A -85,B 0,C 180,E1 27874.577,E2 27874.577} C_VEL
LIN {X 0,Y 592.911,Z 206.4,A -85,B 0,C 180,E1 27871.769,E2 27871.769} C_VEL
LIN {X 0,Y 592.806,Z 180.071,A -85,B 0,C 180,E1 27869.49,E2 27869.49} C_VEL
LIN {X 0,Y 592.568,Z 170.076,A -85,B 0,C 180,E1 27868.627,E2 27868.627} C_VEL
LIN {X 0,Y 592.039,Z 167.993,A -85,B 0,C 180,E1 27868.401,E2 27868.401} C_VEL
LIN {X 0,Y 592.033,Z 167.987,A -85,B 0,C 180,E1 27865.073,E2 27865.073} C_VEL
LIN {X 0,Y 591.998,Z 167.99,A -85,B 0,C 180,E1 27861.912,E2 27861.912} C_VEL
LIN {X 0,Y 592.017,Z 168.18,A -85,B 0,C 180,E1 27860.135,E2 27860.135} C_VEL
LIN {X 0,Y 593.41,Z 171.639,A -85,B 0,C 180,E1 27859.998,E2 27859.998} C_VEL
LIN {X 0,Y 594.39,Z 173.379,A -85,B 0,C 180,E1 27859.912,E2 27859.912} C_VEL
LIN {X 0,Y 593.936,Z 399.835,A -85,B 0,C 180,E1 27856.797,E2 27856.797} C_VEL
LIN {X 0,Y 593.825,Z 463.318,A -85,B 0,C 180,E1 27855.908,E2 27855.908} C_VEL
LIN {X 0,Y 593.694,Z 484.376,A -85,B 0,C 180,E1 27855.43,E2 27855.43} C_VEL
LIN {X 0,Y 593.51,Z 505.977,A -85,B 0,C 180,E1 27854.764,E2 27854.764} C_VEL
LIN {X 0,Y 593.384,Z 526.027,A -85,B 0,C 180,E1 27853.966,E2 27853.966} C_VEL
LIN {X 0,Y 593.176,Z 546.098,A -85,B 0,C 180,E1 27852.983,E2 27852.983} C_VEL
LIN {X 0,Y 592.968,Z 566.034,A -85,B 0,C 180,E1 27851.815,E2 27851.815} C_VEL
LIN {X 0,Y 592.775,Z 585.857,A -85,B 0,C 180,E1 27850.433,E2 27850.433} C_VEL
LIN {X 0,Y 592.584,Z 603.306,A -85,B 0,C 180,E1 27849.003,E2 27849.003} C_VEL
LIN {X 0,Y 592.414,Z 620.071,A -85,B 0,C 180,E1 27847.416,E2 27847.416} C_VEL
LIN {X 0,Y 592.259,Z 636.37,A -85,B 0,C 180,E1 27845.622,E2 27845.622} C_VEL
LIN {X 0,Y 592.144,Z 650.439,A -85,B 0,C 180,E1 27843.822,E2 27843.822} C_VEL
LIN {X 0,Y 592.068,Z 662.504,A -85,B 0,C 180,E1 27842.024,E2 27842.024} C_VEL
LIN {X 0,Y 591.999,Z 673.44,A -85,B 0,C 180,E1 27840.107,E2 27840.107} C_VEL
LIN {X 0,Y 591.96,Z 683.01,A -85,B 0,C 180,E1 27838.116,E2 27838.116} C_VEL
LIN {X 0,Y 591.939,Z 690.637,A -85,B 0,C 180,E1 27836.159,E2 27836.159} C_VEL
LIN {X 0,Y 591.923,Z 697.188,A -85,B 0,C 180,E1 27834.022,E2 27834.022} C_VEL
LIN {X 0,Y 591.915,Z 701.864,A -85,B 0,C 180,E1 27831.971,E2 27831.971} C_VEL
LIN {X 0,Y 591.904,Z 704.914,A -85,B 0,C 180,E1 27829.849,E2 27829.849} C_VEL
LIN {X 0,Y 591.9,Z 706.339,A -85,B 0,C 180,E1 27827.686,E2 27827.686} C_VEL
LIN {X 0,Y 591.905,Z 706.193,A -85,B 0,C 180,E1 27825.663,E2 27825.663} C_VEL
LIN {X 0,Y 591.917,Z 704.357,A -85,B 0,C 180,E1 27823.58,E2 27823.58} C_VEL
LIN {X 0,Y 591.918,Z 700.749,A -85,B 0,C 180,E1 27821.399,E2 27821.399} C_VEL
LIN {X 0,Y 591.917,Z 695.723,A -85,B 0,C 180,E1 27819.333,E2 27819.333} C_VEL
LIN {X 0,Y 591.925,Z 689.281,A -85,B 0,C 180,E1 27817.376,E2 27817.376} C_VEL
LIN {X 0,Y 591.956,Z 680.932,A -85,B 0,C 180,E1 27815.331,E2 27815.331} C_VEL
LIN {X 0,Y 592.003,Z 671.28,A -85,B 0,C 180,E1 27813.389,E2 27813.389} C_VEL
LIN {X 0,Y 592.071,Z 659.727,A -85,B 0,C 180,E1 27811.452,E2 27811.452} C_VEL
LIN {X 0,Y 592.177,Z 646.176,A -85,B 0,C 180,E1 27809.516,E2 27809.516} C_VEL
LIN {X 0,Y 592.32,Z 632.022,A -85,B 0,C 180,E1 27807.775,E2 27807.775} C_VEL
LIN {X 0,Y 592.47,Z 615.51,A -85,B 0,C 180,E1 27806.033,E2 27806.033} C_VEL
LIN {X 0,Y 592.623,Z 598.373,A -85,B 0,C 180,E1 27804.482,E2 27804.482} C_VEL
LIN {X 0,Y 592.82,Z 579.677,A -85,B 0,C 180,E1 27803.025,E2 27803.025} C_VEL
LIN {X 0,Y 593.046,Z 559.854,A -85,B 0,C 180,E1 27801.712,E2 27801.712} C_VEL
LIN {X 0,Y 593.258,Z 539.735,A -85,B 0,C 180,E1 27800.591,E2 27800.591} C_VEL
LIN {X 0,Y 593.404,Z 520.542,A -85,B 0,C 180,E1 27799.712,E2 27799.712} C_VEL
LIN {X 0,Y 593.59,Z 499.231,A -85,B 0,C 180,E1 27798.917,E2 27798.917} C_VEL
LIN {X 0,Y 593.728,Z 478.115,A -85,B 0,C 180,E1 27798.317,E2 27798.317} C_VEL
LIN {X 0,Y 593.833,Z 456.779,A -85,B 0,C 180,E1 27797.897,E2 27797.897} C_VEL
LIN {X 0,Y 594.18,Z 241.684,A -85,B 0,C 180,E1 27794.943,E2 27794.943} C_VEL
LIN {X 0,Y 594.223,Z 172.674,A -85,B 0,C 180,E1 27793.977,E2 27793.977} C_VEL
LIN {X 0,Y 592.286,Z 169.437,A -85,B 0,C 180,E1 27793.81,E2 27793.81} C_VEL
LIN {X 0,Y 591.971,Z 167.996,A -85,B 0,C 180,E1 27793.745,E2 27793.745} C_VEL
LIN {X 0,Y 592,Z 167.99,A -85,B 0,C 180,E1 27790.463,E2 27790.463} C_VEL
LIN {X 0,Y 592.034,Z 167.99,A -85,B 0,C 180,E1 27787.353,E2 27787.353} C_VEL
LIN {X 0,Y 592.031,Z 167.992,A -85,B 0,C 180,E1 27784.061,E2 27784.061} C_VEL
LIN {X 0,Y 592.038,Z 167.985,A -85,B 0,C 180,E1 27780.786,E2 27780.786} C_VEL
LIN {X 0,Y 591.984,Z 167.99,A -85,B 0,C 180,E1 27777.619,E2 27777.619} C_VEL
LIN {X 0,Y 592.002,Z 167.993,A -85,B 0,C 180,E1 27774.479,E2 27774.479} C_VEL
LIN {X 0,Y 591.998,Z 167.991,A -85,B 0,C 180,E1 27771.444,E2 27771.444} C_VEL
LIN {X 0,Y 592.004,Z 167.986,A -85,B 0,C 180,E1 27768.284,E2 27768.284} C_VEL
LIN {X 0,Y 592.028,Z 167.985,A -85,B 0,C 180,E1 27765.094,E2 27765.094} C_VEL
LIN {X 0,Y 592.031,Z 167.991,A -85,B 0,C 180,E1 27761.844,E2 27761.844} C_VEL
LIN {X 0,Y 592.038,Z 167.988,A -85,B 0,C 180,E1 27758.549,E2 27758.549} C_VEL
LIN {X 0,Y 591.973,Z 167.991,A -85,B 0,C 180,E1 27755.5,E2 27755.5} C_VEL
LIN {X 0,Y 591.99,Z 167.99,A -85,B 0,C 180,E1 27752.257,E2 27752.257} C_VEL
LIN {X 0,Y 592.03,Z 167.993,A -85,B 0,C 180,E1 27749.174,E2 27749.174} C_VEL
LIN {X 0,Y 592.01,Z 167.989,A -85,B 0,C 180,E1 27745.941,E2 27745.941} C_VEL
LIN {X 0,Y 592.04,Z 167.981,A -85,B 0,C 180,E1 27742.648,E2 27742.648} C_VEL
LIN {X 0,Y 592.004,Z 167.989,A -85,B 0,C 180,E1 27739.434,E2 27739.434} C_VEL
LIN {X 0,Y 592.034,Z 167.993,A -85,B 0,C 180,E1 27736.281,E2 27736.281} C_VEL
LIN {X 0,Y 591.976,Z 167.991,A -85,B 0,C 180,E1 27733.181,E2 27733.181} C_VEL
LIN {X 0,Y 591.985,Z 167.99,A -85,B 0,C 180,E1 27729.921,E2 27729.921} C_VEL
LIN {X 0,Y 592.035,Z 167.988,A -85,B 0,C 180,E1 27726.79,E2 27726.79} C_VEL
LIN {X 0,Y 592.033,Z 167.991,A -85,B 0,C 180,E1 27723.486,E2 27723.486} C_VEL
LIN {X 0,Y 592.031,Z 167.987,A -85,B 0,C 180,E1 27720.194,E2 27720.194} C_VEL
LIN {X 0,Y 591.994,Z 167.989,A -85,B 0,C 180,E1 27717.096,E2 27717.096} C_VEL
LIN {X 0,Y 591.989,Z 167.993,A -85,B 0,C 180,E1 27713.892,E2 27713.892} C_VEL
LIN {X 0,Y 592.004,Z 167.992,A -85,B 0,C 180,E1 27710.865,E2 27710.865} C_VEL
LIN {X 0,Y 591.993,Z 167.989,A -85,B 0,C 180,E1 27707.713,E2 27707.713} C_VEL
LIN {X 0,Y 592.033,Z 167.986,A -85,B 0,C 180,E1 27704.624,E2 27704.624} C_VEL
LIN {X 0,Y 592.027,Z 167.992,A -85,B 0,C 180,E1 27701.284,E2 27701.284} C_VEL
LIN {X 0,Y 592.035,Z 167.987,A -85,B 0,C 180,E1 27698.085,E2 27698.085} C_VEL
LIN {X 0,Y 591.985,Z 167.991,A -85,B 0,C 180,E1 27695.024,E2 27695.024} C_VEL
LIN {X 0,Y 591.979,Z 167.993,A -85,B 0,C 180,E1 27691.776,E2 27691.776} C_VEL
LIN {X 0,Y 592.027,Z 167.992,A -85,B 0,C 180,E1 27688.712,E2 27688.712} C_VEL
LIN {X 0,Y 592.004,Z 167.992,A -85,B 0,C 180,E1 27685.508,E2 27685.508} C_VEL
LIN {X 0,Y 592.055,Z 168.192,A -85,B 0,C 180,E1 27682.649,E2 27682.649} C_VEL
LIN {X 0,Y 593.342,Z 171.467,A -85,B 0,C 180,E1 27682.288,E2 27682.288} C_VEL
LIN {X 0,Y 594.887,Z 175.244,A -85,B 0,C 180,E1 27681.868,E2 27681.868} C_VEL
LIN {X 0,Y 594.518,Z 216.556,A -85,B 0,C 180,E1 27678.885,E2 27678.885} C_VEL
LIN {X 0,Y 594.628,Z 259.353,A -85,B 0,C 180,E1 27675.883,E2 27675.883} C_VEL
LIN {X 0,Y 596.272,Z 269.237,A -85,B 0,C 180,E1 27675.094,E2 27675.094} C_VEL
LIN {X 0,Y 598.276,Z 275.248,A -85,B 0,C 180,E1 27674.47,E2 27674.47} C_VEL
LIN {X 0,Y 600.057,Z 278.571,A -85,B 0,C 180,E1 27673.881,E2 27673.881} C_VEL
LIN {X 0,Y 601.343,Z 279.768,A -85,B 0,C 180,E1 27673.369,E2 27673.369} C_VEL
LIN {X 0,Y 602.272,Z 279.355,A -85,B 0,C 180,E1 27672.796,E2 27672.796} C_VEL
LIN {X 0,Y 602.419,Z 277.22,A -85,B 0,C 180,E1 27672.265,E2 27672.265} C_VEL
LIN {X 0,Y 601.755,Z 273.457,A -85,B 0,C 180,E1 27671.813,E2 27671.813} C_VEL
LIN {X 0,Y 600.444,Z 268.39,A -85,B 0,C 180,E1 27671.484,E2 27671.484} C_VEL
LIN {X 0,Y 598.609,Z 260.934,A -85,B 0,C 180,E1 27671.258,E2 27671.258} C_VEL
LIN {X 0,Y 597.468,Z 250.833,A -85,B 0,C 180,E1 27671.133,E2 27671.133} C_VEL
LIN {X 0,Y 597.28,Z 227.658,A -85,B 0,C 180,E1 27671.113,E2 27671.113} C_VEL
LIN {X 0,Y 597.169,Z 175.564,A -85,B 0,C 180,E1 27671.101,E2 27671.101} C_VEL
LIN {X 0,Y 596.103,Z 174.027,A -85,B 0,C 180,E1 27670.983,E2 27670.983} C_VEL
LIN {X 0,Y 593.405,Z 171.618,A -85,B 0,C 180,E1 27670.682,E2 27670.682} C_VEL
LIN {X 0,Y 592.104,Z 168.573,A -85,B 0,C 180,E1 27670.536,E2 27670.536} C_VEL
LIN {X 0,Y 592.012,Z 167.994,A -85,B 0,C 180,E1 27670.517,E2 27670.517} C_VEL
LIN {X 0,Y 592.039,Z 168.013,A -85,B 0,C 180,E1 27667.383,E2 27667.383} C_VEL
LIN {X 0,Y 594.192,Z 174.392,A -85,B 0,C 180,E1 27666.777,E2 27666.777} C_VEL
LIN {X 0,Y 593.831,Z 219.326,A -85,B 0,C 180,E1 27663.72,E2 27663.72} C_VEL
LIN {X 0,Y 593.878,Z 227.214,A -85,B 0,C 180,E1 27663.218,E2 27663.218} C_VEL
LIN {X 0,Y 594.403,Z 231.519,A -85,B 0,C 180,E1 27663.124,E2 27663.124} C_VEL
LIN {X 0,Y 593.979,Z 449.731,A -85,B 0,C 180,E1 27660.115,E2 27660.115} C_VEL
LIN {X 0,Y 593.826,Z 532.792,A -85,B 0,C 180,E1 27658.962,E2 27658.962} C_VEL
LIN {X 0,Y 593.699,Z 554.492,A -85,B 0,C 180,E1 27658.473,E2 27658.473} C_VEL
LIN {X 0,Y 593.528,Z 576.529,A -85,B 0,C 180,E1 27657.789,E2 27657.789} C_VEL
LIN {X 0,Y 593.371,Z 597.417,A -85,B 0,C 180,E1 27656.952,E2 27656.952} C_VEL
LIN {X 0,Y 593.173,Z 616.751,A -85,B 0,C 180,E1 27655.993,E2 27655.993} C_VEL
LIN {X 0,Y 592.955,Z 636.539,A -85,B 0,C 180,E1 27654.826,E2 27654.826} C_VEL
LIN {X 0,Y 592.784,Z 655.704,A -85,B 0,C 180,E1 27653.49,E2 27653.49} C_VEL
LIN {X 0,Y 592.582,Z 674.234,A -85,B 0,C 180,E1 27651.97,E2 27651.97} C_VEL
LIN {X 0,Y 592.408,Z 691.208,A -85,B 0,C 180,E1 27650.346,E2 27650.346} C_VEL
LIN {X 0,Y 592.257,Z 706.874,A -85,B 0,C 180,E1 27648.607,E2 27648.607} C_VEL
LIN {X 0,Y 592.134,Z 721.052,A -85,B 0,C 180,E1 27646.781,E2 27646.781} C_VEL
LIN {X 0,Y 592.054,Z 733.746,A -85,B 0,C 180,E1 27644.874,E2 27644.874} C_VEL
LIN {X 0,Y 591.992,Z 744.453,A -85,B 0,C 180,E1 27642.958,E2 27642.958} C_VEL
LIN {X 0,Y 591.946,Z 754.072,A -85,B 0,C 180,E1 27640.905,E2 27640.905} C_VEL
LIN {X 0,Y 591.936,Z 761.599,A -85,B 0,C 180,E1 27638.94,E2 27638.94} C_VEL
LIN {X 0,Y 591.925,Z 767.66,A -85,B 0,C 180,E1 27636.888,E2 27636.888} C_VEL
LIN {X 0,Y 591.916,Z 772.367,A -85,B 0,C 180,E1 27634.713,E2 27634.713} C_VEL
LIN {X 0,Y 591.907,Z 775.239,A -85,B 0,C 180,E1 27632.614,E2 27632.614} C_VEL
LIN {X 0,Y 591.897,Z 776.379,A -85,B 0,C 180,E1 27630.581,E2 27630.581} C_VEL
LIN {X 0,Y 591.898,Z 776.018,A -85,B 0,C 180,E1 27628.451,E2 27628.451} C_VEL
LIN {X 0,Y 591.903,Z 774.116,A -85,B 0,C 180,E1 27626.416,E2 27626.416} C_VEL
LIN {X 0,Y 591.918,Z 770.608,A -85,B 0,C 180,E1 27624.377,E2 27624.377} C_VEL
LIN {X 0,Y 591.921,Z 765.586,A -85,B 0,C 180,E1 27622.331,E2 27622.331} C_VEL
LIN {X 0,Y 591.922,Z 759.114,A -85,B 0,C 180,E1 27620.373,E2 27620.373} C_VEL
LIN {X 0,Y 591.955,Z 750.604,A -85,B 0,C 180,E1 27618.306,E2 27618.306} C_VEL
LIN {X 0,Y 592.01,Z 740.689,A -85,B 0,C 180,E1 27616.323,E2 27616.323} C_VEL
LIN {X 0,Y 592.07,Z 729.266,A -85,B 0,C 180,E1 27614.424,E2 27614.424} C_VEL
LIN {X 0,Y 592.186,Z 715.79,A -85,B 0,C 180,E1 27612.51,E2 27612.51} C_VEL
LIN {X 0,Y 592.316,Z 701.672,A -85,B 0,C 180,E1 27610.781,E2 27610.781} C_VEL
LIN {X 0,Y 592.468,Z 685.714,A -85,B 0,C 180,E1 27609.097,E2 27609.097} C_VEL
LIN {X 0,Y 592.633,Z 668.197,A -85,B 0,C 180,E1 27607.51,E2 27607.51} C_VEL
LIN {X 0,Y 592.818,Z 649.869,A -85,B 0,C 180,E1 27606.084,E2 27606.084} C_VEL
LIN {X 0,Y 593.042,Z 630.641,A -85,B 0,C 180,E1 27604.804,E2 27604.804} C_VEL
LIN {X 0,Y 593.237,Z 610.757,A -85,B 0,C 180,E1 27603.687,E2 27603.687} C_VEL
LIN {X 0,Y 593.407,Z 591.054,A -85,B 0,C 180,E1 27602.776,E2 27602.776} C_VEL
LIN {X 0,Y 593.599,Z 569.633,A -85,B 0,C 180,E1 27601.976,E2 27601.976} C_VEL
LIN {X 0,Y 593.725,Z 548.586,A -85,B 0,C 180,E1 27601.372,E2 27601.372} C_VEL
LIN {X 0,Y 593.838,Z 527.009,A -85,B 0,C 180,E1 27600.945,E2 27600.945} C_VEL
LIN {X 0,Y 594.288,Z 290.149,A -85,B 0,C 180,E1 27597.694,E2 27597.694} C_VEL
LIN {X 0,Y 594.217,Z 225.903,A -85,B 0,C 180,E1 27596.785,E2 27596.785} C_VEL
LIN {X 0,Y 594.128,Z 216.664,A -85,B 0,C 180,E1 27596.38,E2 27596.38} C_VEL
LIN {X 0,Y 594.328,Z 173.706,A -85,B 0,C 180,E1 27594.347,E2 27594.347} C_VEL
LIN {X 0,Y 592.087,Z 168.369,A -85,B 0,C 180,E1 27593.932,E2 27593.932} C_VEL
LIN {X 0,Y 592.033,Z 167.987,A -85,B 0,C 180,E1 27593.884,E2 27593.884} C_VEL
LIN {X 0,Y 592.014,Z 167.992,A -85,B 0,C 180,E1 27590.671,E2 27590.671} C_VEL
LIN {X 0,Y 592.057,Z 168.183,A -85,B 0,C 180,E1 27589.47,E2 27589.47} C_VEL
LIN {X 0,Y 593.163,Z 171.205,A -85,B 0,C 180,E1 27589.345,E2 27589.345} C_VEL
LIN {X 0,Y 595.613,Z 173.709,A -85,B 0,C 180,E1 27589.071,E2 27589.071} C_VEL
LIN {X 0,Y 596.679,Z 174.677,A -85,B 0,C 180,E1 27588.953,E2 27588.953} C_VEL
LIN {X 0,Y 599.298,Z 178.187,A -85,B 0,C 180,E1 27588.648,E2 27588.648} C_VEL
LIN {X 0,Y 601.735,Z 180.319,A -85,B 0,C 180,E1 27588.217,E2 27588.217} C_VEL
LIN {X 0,Y 603.525,Z 181.348,A -85,B 0,C 180,E1 27587.636,E2 27587.636} C_VEL
LIN {X 0,Y 603.804,Z 182.026,A -85,B 0,C 180,E1 27587.327,E2 27587.327} C_VEL
LIN {X 0,Y 603.381,Z 182.866,A -85,B 0,C 180,E1 27586.812,E2 27586.812} C_VEL
LIN {X 0,Y 602.386,Z 182.22,A -85,B 0,C 180,E1 27586.331,E2 27586.331} C_VEL
LIN {X 0,Y 600.752,Z 180.298,A -85,B 0,C 180,E1 27585.834,E2 27585.834} C_VEL
LIN {X 0,Y 597.644,Z 178.061,A -85,B 0,C 180,E1 27585.318,E2 27585.318} C_VEL
LIN {X 0,Y 594.829,Z 174.339,A -85,B 0,C 180,E1 27584.909,E2 27584.909} C_VEL
LIN {X 0,Y 592.274,Z 169.286,A -85,B 0,C 180,E1 27584.474,E2 27584.474} C_VEL
LIN {X 0,Y 592.003,Z 167.992,A -85,B 0,C 180,E1 27584.364,E2 27584.364} C_VEL
LIN {X 0,Y 592.041,Z 167.99,A -85,B 0,C 180,E1 27581.129,E2 27581.129} C_VEL
LIN {X 0,Y 592.028,Z 167.984,A -85,B 0,C 180,E1 27577.811,E2 27577.811} C_VEL
LIN {X 0,Y 591.991,Z 167.99,A -85,B 0,C 180,E1 27574.576,E2 27574.576} C_VEL
LIN {X 0,Y 592.039,Z 167.991,A -85,B 0,C 180,E1 27571.456,E2 27571.456} C_VEL
LIN {X 0,Y 592.025,Z 168.211,A -85,B 0,C 180,E1 27570.835,E2 27570.835} C_VEL
LIN {X 0,Y 592.627,Z 194.842,A -85,B 0,C 180,E1 27568.795,E2 27568.795} C_VEL
LIN {X 0,Y 592.882,Z 219.172,A -85,B 0,C 180,E1 27566.821,E2 27566.821} C_VEL
LIN {X 0,Y 592.695,Z 256.252,A -85,B 0,C 180,E1 27563.648,E2 27563.648} C_VEL
LIN {X 0,Y 592.483,Z 292.418,A -85,B 0,C 180,E1 27560.624,E2 27560.624} C_VEL
LIN {X 0,Y 592.425,Z 312.982,A -85,B 0,C 180,E1 27558.956,E2 27558.956} C_VEL
LIN {X 0,Y 592.681,Z 327.873,A -85,B 0,C 180,E1 27558.76,E2 27558.76} C_VEL
LIN {X 0,Y 592.526,Z 482.113,A -85,B 0,C 180,E1 27556.815,E2 27556.815} C_VEL
LIN {X 0,Y 592.501,Z 499.878,A -85,B 0,C 180,E1 27556.403,E2 27556.403} C_VEL
LIN {X 0,Y 592.433,Z 516.996,A -85,B 0,C 180,E1 27555.817,E2 27555.817} C_VEL
LIN {X 0,Y 592.345,Z 533.236,A -85,B 0,C 180,E1 27555.067,E2 27555.067} C_VEL
LIN {X 0,Y 592.255,Z 548.425,A -85,B 0,C 180,E1 27554.169,E2 27554.169} C_VEL
LIN {X 0,Y 592.164,Z 562.605,A -85,B 0,C 180,E1 27553.126,E2 27553.126} C_VEL
LIN {X 0,Y 592.089,Z 576.322,A -85,B 0,C 180,E1 27551.889,E2 27551.889} C_VEL
LIN {X 0,Y 592.027,Z 587.962,A -85,B 0,C 180,E1 27550.602,E2 27550.602} C_VEL
LIN {X 0,Y 591.972,Z 598.698,A -85,B 0,C 180,E1 27549.135,E2 27549.135} C_VEL
LIN {X 0,Y 591.947,Z 607.846,A -85,B 0,C 180,E1 27547.57,E2 27547.57} C_VEL
LIN {X 0,Y 591.927,Z 614.938,A -85,B 0,C 180,E1 27546.011,E2 27546.011} C_VEL
LIN {X 0,Y 591.92,Z 620.464,A -85,B 0,C 180,E1 27544.359,E2 27544.359} C_VEL
LIN {X 0,Y 591.914,Z 624.137,A -85,B 0,C 180,E1 27542.711,E2 27542.711} C_VEL
LIN {X 0,Y 591.91,Z 626.158,A -85,B 0,C 180,E1 27540.968,E2 27540.968} C_VEL
LIN {X 0,Y 591.914,Z 626.335,A -85,B 0,C 180,E1 27539.225,E2 27539.225} C_VEL
LIN {X 0,Y 591.915,Z 624.597,A -85,B 0,C 180,E1 27537.482,E2 27537.482} C_VEL
LIN {X 0,Y 591.915,Z 620.947,A -85,B 0,C 180,E1 27535.737,E2 27535.737} C_VEL
LIN {X 0,Y 591.922,Z 615.653,A -85,B 0,C 180,E1 27534.085,E2 27534.085} C_VEL
LIN {X 0,Y 591.946,Z 608.82,A -85,B 0,C 180,E1 27532.527,E2 27532.527} C_VEL
LIN {X 0,Y 591.974,Z 599.921,A -85,B 0,C 180,E1 27530.962,E2 27530.962} C_VEL
LIN {X 0,Y 591.983,Z 597.495,A -85,B 0,C 180,E1 27530.591,E2 27530.591} C_VEL
LIN {X 0,Y 591.035,Z 593.272,A -85,B 0,C 180,E1 27529.967,E2 27529.967} C_VEL
LIN {X 0,Y 586.314,Z 584.534,A -85,B 0,C 180,E1 27528.786,E2 27528.786} C_VEL
LIN {X 0,Y 584.364,Z 578.941,A -85,B 0,C 180,E1 27528.132,E2 27528.132} C_VEL
LIN {X 0,Y 584.179,Z 576.67,A -85,B 0,C 180,E1 27527.893,E2 27527.893} C_VEL
LIN {X 0,Y 584.288,Z 563.688,A -85,B 0,C 180,E1 27526.693,E2 27526.693} C_VEL
LIN {X 0,Y 584.43,Z 548.93,A -85,B 0,C 180,E1 27525.581,E2 27525.581} C_VEL
LIN {X 0,Y 584.574,Z 533.035,A -85,B 0,C 180,E1 27524.626,E2 27524.626} C_VEL
LIN {X 0,Y 584.686,Z 516.703,A -85,B 0,C 180,E1 27523.865,E2 27523.865} C_VEL
LIN {X 0,Y 584.815,Z 499.418,A -85,B 0,C 180,E1 27523.272,E2 27523.272} C_VEL
LIN {X 0,Y 584.903,Z 481.749,A -85,B 0,C 180,E1 27522.862,E2 27522.862} C_VEL
LIN {X 0,Y 584.973,Z 314.55,A -85,B 0,C 180,E1 27520.723,E2 27520.723} C_VEL
LIN {X 0,Y 584.68,Z 312.534,A -85,B 0,C 180,E1 27520.671,E2 27520.671} C_VEL
LIN {X 0,Y 584.917,Z 276.146,A -85,B 0,C 180,E1 27517.543,E2 27517.543} C_VEL
LIN {X 0,Y 585.204,Z 239.529,A -85,B 0,C 180,E1 27514.334,E2 27514.334} C_VEL
LIN {X 0,Y 585.398,Z 205.29,A -85,B 0,C 180,E1 27511.318,E2 27511.318} C_VEL
LIN {X 0,Y 585.108,Z 172.807,A -85,B 0,C 180,E1 27508.509,E2 27508.509} C_VEL
LIN {X 0,Y 584.086,Z 168.983,A -85,B 0,C 180,E1 27508.111,E2 27508.111} C_VEL
LIN {X 0,Y 584.092,Z 168.979,A -85,B 0,C 180,E1 27504.888,E2 27504.888} C_VEL
LIN {X 0,Y 584.065,Z 168.979,A -85,B 0,C 180,E1 27501.705,E2 27501.705} C_VEL
LIN {X 0,Y 584.112,Z 169.182,A -85,B 0,C 180,E1 27500.629,E2 27500.629} C_VEL
LIN {X 0,Y 585.453,Z 172.578,A -85,B 0,C 180,E1 27500.493,E2 27500.493} C_VEL
LIN {X 0,Y 587.664,Z 176.426,A -85,B 0,C 180,E1 27500.295,E2 27500.295} C_VEL
LIN {X 0,Y 586.988,Z 401.989,A -85,B 0,C 180,E1 27497.157,E2 27497.157} C_VEL
LIN {X 0,Y 586.816,Z 463.421,A -85,B 0,C 180,E1 27496.285,E2 27496.285} C_VEL
LIN {X 0,Y 586.62,Z 484.558,A -85,B 0,C 180,E1 27495.8,E2 27495.8} C_VEL
LIN {X 0,Y 586.359,Z 505.891,A -85,B 0,C 180,E1 27495.137,E2 27495.137} C_VEL
LIN {X 0,Y 586.148,Z 526.427,A -85,B 0,C 180,E1 27494.31,E2 27494.31} C_VEL
LIN {X 0,Y 585.835,Z 546.306,A -85,B 0,C 180,E1 27493.323,E2 27493.323} C_VEL
LIN {X 0,Y 585.539,Z 566.057,A -85,B 0,C 180,E1 27492.151,E2 27492.151} C_VEL
LIN {X 0,Y 585.23,Z 586.011,A -85,B 0,C 180,E1 27490.741,E2 27490.741} C_VEL
LIN {X 0,Y 584.938,Z 603.436,A -85,B 0,C 180,E1 27489.295,E2 27489.295} C_VEL
LIN {X 0,Y 584.671,Z 620.778,A -85,B 0,C 180,E1 27487.627,E2 27487.627} C_VEL
LIN {X 0,Y 584.443,Z 636.514,A -85,B 0,C 180,E1 27485.864,E2 27485.864} C_VEL
LIN {X 0,Y 584.269,Z 651.042,A -85,B 0,C 180,E1 27483.969,E2 27483.969} C_VEL
LIN {X 0,Y 584.153,Z 662.944,A -85,B 0,C 180,E1 27482.163,E2 27482.163} C_VEL
LIN {X 0,Y 584.045,Z 674.064,A -85,B 0,C 180,E1 27480.169,E2 27480.169} C_VEL
LIN {X 0,Y 583.978,Z 683.75,A -85,B 0,C 180,E1 27478.089,E2 27478.089} C_VEL
LIN {X 0,Y 583.95,Z 691.277,A -85,B 0,C 180,E1 27476.107,E2 27476.107} C_VEL
LIN {X 0,Y 583.927,Z 697.369,A -85,B 0,C 180,E1 27474.05,E2 27474.05} C_VEL
LIN {X 0,Y 583.918,Z 701.889,A -85,B 0,C 180,E1 27472.025,E2 27472.025} C_VEL
LIN {X 0,Y 583.908,Z 704.877,A -85,B 0,C 180,E1 27469.923,E2 27469.923} C_VEL
LIN {X 0,Y 583.901,Z 706.327,A -85,B 0,C 180,E1 27467.747,E2 27467.747} C_VEL
LIN {X 0,Y 583.906,Z 706.213,A -85,B 0,C 180,E1 27465.697,E2 27465.697} C_VEL
LIN {X 0,Y 583.916,Z 704.398,A -85,B 0,C 180,E1 27463.568,E2 27463.568} C_VEL
LIN {X 0,Y 583.919,Z 700.823,A -85,B 0,C 180,E1 27461.357,E2 27461.357} C_VEL
LIN {X 0,Y 583.925,Z 695.824,A -85,B 0,C 180,E1 27459.263,E2 27459.263} C_VEL
LIN {X 0,Y 583.94,Z 689.409,A -85,B 0,C 180,E1 27457.28,E2 27457.28} C_VEL
LIN {X 0,Y 583.99,Z 681.105,A -85,B 0,C 180,E1 27455.206,E2 27455.206} C_VEL
LIN {X 0,Y 584.068,Z 670.96,A -85,B 0,C 180,E1 27453.14,E2 27453.14} C_VEL
LIN {X 0,Y 584.158,Z 659.974,A -85,B 0,C 180,E1 27451.275,E2 27451.275} C_VEL
LIN {X 0,Y 584.32,Z 646.475,A -85,B 0,C 180,E1 27449.314,E2 27449.314} C_VEL
LIN {X 0,Y 584.528,Z 632.367,A -85,B 0,C 180,E1 27447.549,E2 27447.549} C_VEL
LIN {X 0,Y 584.775,Z 615.408,A -85,B 0,C 180,E1 27445.735,E2 27445.735} C_VEL
LIN {X 0,Y 585.006,Z 598.827,A -85,B 0,C 180,E1 27444.213,E2 27444.213} C_VEL
LIN {X 0,Y 585.297,Z 580.221,A -85,B 0,C 180,E1 27442.738,E2 27442.738} C_VEL
LIN {X 0,Y 585.627,Z 561.316,A -85,B 0,C 180,E1 27441.458,E2 27441.458} C_VEL
LIN {X 0,Y 585.953,Z 540.485,A -85,B 0,C 180,E1 27440.274,E2 27440.274} C_VEL
LIN {X 0,Y 586.178,Z 521.398,A -85,B 0,C 180,E1 27439.385,E2 27439.385} C_VEL
LIN {X 0,Y 586.462,Z 500.549,A -85,B 0,C 180,E1 27438.587,E2 27438.587} C_VEL
LIN {X 0,Y 586.663,Z 479.095,A -85,B 0,C 180,E1 27437.965,E2 27437.965} C_VEL
LIN {X 0,Y 586.83,Z 457.34,A -85,B 0,C 180,E1 27437.525,E2 27437.525} C_VEL
LIN {X 0,Y 587.391,Z 242.665,A -85,B 0,C 180,E1 27434.542,E2 27434.542} C_VEL
LIN {X 0,Y 587.447,Z 176.017,A -85,B 0,C 180,E1 27433.595,E2 27433.595} C_VEL
LIN {X 0,Y 584.289,Z 170.1,A -85,B 0,C 180,E1 27433.306,E2 27433.306} C_VEL
LIN {X 0,Y 584.075,Z 168.984,A -85,B 0,C 180,E1 27433.26,E2 27433.26} C_VEL
LIN {X 0,Y 584.054,Z 168.98,A -85,B 0,C 180,E1 27430.082,E2 27430.082} C_VEL
LIN {X 0,Y 584.1,Z 168.973,A -85,B 0,C 180,E1 27426.921,E2 27426.921} C_VEL
LIN {X 0,Y 584.082,Z 168.979,A -85,B 0,C 180,E1 27423.572,E2 27423.572} C_VEL
LIN {X 0,Y 584.097,Z 168.979,A -85,B 0,C 180,E1 27420.349,E2 27420.349} C_VEL
LIN {X 0,Y 584.061,Z 168.978,A -85,B 0,C 180,E1 27417.199,E2 27417.199} C_VEL
LIN {X 0,Y 584.027,Z 168.982,A -85,B 0,C 180,E1 27413.908,E2 27413.908} C_VEL
LIN {X 0,Y 584.1,Z 168.978,A -85,B 0,C 180,E1 27410.828,E2 27410.828} C_VEL
LIN {X 0,Y 584.089,Z 168.979,A -85,B 0,C 180,E1 27407.545,E2 27407.545} C_VEL
LIN {X 0,Y 584.081,Z 168.974,A -85,B 0,C 180,E1 27404.302,E2 27404.302} C_VEL
LIN {X 0,Y 584.076,Z 168.974,A -85,B 0,C 180,E1 27401.099,E2 27401.099} C_VEL
LIN {X 0,Y 584.057,Z 168.979,A -85,B 0,C 180,E1 27397.798,E2 27397.798} C_VEL
LIN {X 0,Y 584.093,Z 168.982,A -85,B 0,C 180,E1 27394.575,E2 27394.575} C_VEL
LIN {X 0,Y 584.043,Z 168.979,A -85,B 0,C 180,E1 27391.477,E2 27391.477} C_VEL
LIN {X 0,Y 584.063,Z 168.976,A -85,B 0,C 180,E1 27388.16,E2 27388.16} C_VEL
LIN {X 0,Y 584.09,Z 168.977,A -85,B 0,C 180,E1 27385.013,E2 27385.013} C_VEL
LIN {X 0,Y 584.095,Z 168.981,A -85,B 0,C 180,E1 27381.701,E2 27381.701} C_VEL
LIN {X 0,Y 584.098,Z 168.977,A -85,B 0,C 180,E1 27378.359,E2 27378.359} C_VEL
LIN {X 0,Y 584.039,Z 168.981,A -85,B 0,C 180,E1 27375.287,E2 27375.287} C_VEL
LIN {X 0,Y 584.037,Z 168.981,A -85,B 0,C 180,E1 27371.956,E2 27371.956} C_VEL
LIN {X 0,Y 584.098,Z 168.978,A -85,B 0,C 180,E1 27368.863,E2 27368.863} C_VEL
LIN {X 0,Y 584.072,Z 168.979,A -85,B 0,C 180,E1 27365.699,E2 27365.699} C_VEL
LIN {X 0,Y 584.093,Z 168.974,A -85,B 0,C 180,E1 27362.355,E2 27362.355} C_VEL
LIN {X 0,Y 584.066,Z 168.978,A -85,B 0,C 180,E1 27359.216,E2 27359.216} C_VEL
LIN {X 0,Y 584.081,Z 168.98,A -85,B 0,C 180,E1 27355.976,E2 27355.976} C_VEL
LIN {X 0,Y 584.045,Z 168.982,A -85,B 0,C 180,E1 27352.92,E2 27352.92} C_VEL
LIN {X 0,Y 584.043,Z 168.98,A -85,B 0,C 180,E1 27349.744,E2 27349.744} C_VEL
LIN {X 0,Y 584.098,Z 168.977,A -85,B 0,C 180,E1 27346.639,E2 27346.639} C_VEL
LIN {X 0,Y 584.091,Z 168.981,A -85,B 0,C 180,E1 27343.389,E2 27343.389} C_VEL
LIN {X 0,Y 584.091,Z 168.977,A -85,B 0,C 180,E1 27340.084,E2 27340.084} C_VEL
LIN {X 0,Y 584.059,Z 168.978,A -85,B 0,C 180,E1 27336.92,E2 27336.92} C_VEL
LIN {X 0,Y 584.047,Z 168.981,A -85,B 0,C 180,E1 27333.68,E2 27333.68} C_VEL
LIN {X 0,Y 584.1,Z 168.979,A -85,B 0,C 180,E1 27330.463,E2 27330.463} C_VEL
LIN {X 0,Y 584.06,Z 168.983,A -85,B 0,C 180,E1 27327.251,E2 27327.251} C_VEL
LIN {X 0,Y 584.077,Z 168.98,A -85,B 0,C 180,E1 27323.901,E2 27323.901} C_VEL
LIN {X 0,Y 584.088,Z 168.987,A -85,B 0,C 180,E1 27323.314,E2 27323.314} C_VEL
LIN {X 0,Y 585.423,Z 172.503,A -85,B 0,C 180,E1 27322.923,E2 27322.923} C_VEL
LIN {X 0,Y 588.384,Z 179.01,A -85,B 0,C 180,E1 27322.16,E2 27322.16} C_VEL
LIN {X 0,Y 587.839,Z 220.204,A -85,B 0,C 180,E1 27319.157,E2 27319.157} C_VEL
LIN {X 0,Y 587.789,Z 262.088,A -85,B 0,C 180,E1 27316.186,E2 27316.186} C_VEL
LIN {X 0,Y 589.487,Z 272.731,A -85,B 0,C 180,E1 27315.328,E2 27315.328} C_VEL
LIN {X 0,Y 592.431,Z 280.625,A -85,B 0,C 180,E1 27314.585,E2 27314.585} C_VEL
LIN {X 0,Y 595.089,Z 284.688,A -85,B 0,C 180,E1 27314.019,E2 27314.019} C_VEL
LIN {X 0,Y 597.206,Z 286.627,A -85,B 0,C 180,E1 27313.48,E2 27313.48} C_VEL
LIN {X 0,Y 598.759,Z 287.03,A -85,B 0,C 180,E1 27312.946,E2 27312.946} C_VEL
LIN {X 0,Y 599.66,Z 285.937,A -85,B 0,C 180,E1 27312.384,E2 27312.384} C_VEL
LIN {X 0,Y 599.596,Z 283.277,A -85,B 0,C 180,E1 27311.838,E2 27311.838} C_VEL
LIN {X 0,Y 598.497,Z 279.129,A -85,B 0,C 180,E1 27311.371,E2 27311.371} C_VEL
LIN {X 0,Y 596.55,Z 273.785,A -85,B 0,C 180,E1 27311.033,E2 27311.033} C_VEL
LIN {X 0,Y 594.099,Z 265.772,A -85,B 0,C 180,E1 27310.76,E2 27310.76} C_VEL
LIN {X 0,Y 592.541,Z 255.523,A -85,B 0,C 180,E1 27310.585,E2 27310.585} C_VEL
LIN {X 0,Y 592.054,Z 244.548,A -85,B 0,C 180,E1 27310.53,E2 27310.53} C_VEL
LIN {X 0,Y 592.023,Z 179.919,A -85,B 0,C 180,E1 27310.526,E2 27310.526} C_VEL
LIN {X 0,Y 589.109,Z 176.268,A -85,B 0,C 180,E1 27310.194,E2 27310.194} C_VEL
LIN {X 0,Y 588.304,Z 175.076,A -85,B 0,C 180,E1 27310.101,E2 27310.101} C_VEL
LIN {X 0,Y 585.575,Z 172.755,A -85,B 0,C 180,E1 27309.783,E2 27309.783} C_VEL
LIN {X 0,Y 584.217,Z 169.855,A -85,B 0,C 180,E1 27309.623,E2 27309.623} C_VEL
LIN {X 0,Y 584.059,Z 168.984,A -85,B 0,C 180,E1 27309.588,E2 27309.588} C_VEL
LIN {X 0,Y 584.113,Z 169.148,A -85,B 0,C 180,E1 27307.897,E2 27307.897} C_VEL
LIN {X 0,Y 587.349,Z 177.483,A -85,B 0,C 180,E1 27307.058,E2 27307.058} C_VEL
LIN {X 0,Y 586.824,Z 221.392,A -85,B 0,C 180,E1 27304.036,E2 27304.036} C_VEL
LIN {X 0,Y 586.864,Z 227.22,A -85,B 0,C 180,E1 27303.667,E2 27303.667} C_VEL
LIN {X 0,Y 587.696,Z 232.599,A -85,B 0,C 180,E1 27303.536,E2 27303.536} C_VEL
LIN {X 0,Y 587.054,Z 450.583,A -85,B 0,C 180,E1 27300.496,E2 27300.496} C_VEL
LIN {X 0,Y 586.818,Z 532.791,A -85,B 0,C 180,E1 27299.342,E2 27299.342} C_VEL
LIN {X 0,Y 586.626,Z 554.716,A -85,B 0,C 180,E1 27298.842,E2 27298.842} C_VEL
LIN {X 0,Y 586.366,Z 577.128,A -85,B 0,C 180,E1 27298.136,E2 27298.136} C_VEL
LIN {X 0,Y 586.125,Z 598.089,A -85,B 0,C 180,E1 27297.282,E2 27297.282} C_VEL
LIN {X 0,Y 585.823,Z 617.752,A -85,B 0,C 180,E1 27296.289,E2 27296.289} C_VEL
LIN {X 0,Y 585.486,Z 638.15,A -85,B 0,C 180,E1 27295.057,E2 27295.057} C_VEL
LIN {X 0,Y 585.208,Z 657.349,A -85,B 0,C 180,E1 27293.683,E2 27293.683} C_VEL
LIN {X 0,Y 584.926,Z 675.105,A -85,B 0,C 180,E1 27292.196,E2 27292.196} C_VEL
LIN {X 0,Y 584.66,Z 692.225,A -85,B 0,C 180,E1 27290.523,E2 27290.523} C_VEL
LIN {X 0,Y 584.435,Z 707.727,A -85,B 0,C 180,E1 27288.762,E2 27288.762} C_VEL
LIN {X 0,Y 584.255,Z 721.753,A -85,B 0,C 180,E1 27286.913,E2 27286.913} C_VEL
LIN {X 0,Y 584.13,Z 734.345,A -85,B 0,C 180,E1 27284.979,E2 27284.979} C_VEL
LIN {X 0,Y 584.039,Z 744.856,A -85,B 0,C 180,E1 27283.06,E2 27283.06} C_VEL
LIN {X 0,Y 583.97,Z 754.483,A -85,B 0,C 180,E1 27280.956,E2 27280.956} C_VEL
LIN {X 0,Y 583.941,Z 762.156,A -85,B 0,C 180,E1 27278.896,E2 27278.896} C_VEL
LIN {X 0,Y 583.926,Z 768.171,A -85,B 0,C 180,E1 27276.785,E2 27276.785} C_VEL
LIN {X 0,Y 583.916,Z 772.629,A -85,B 0,C 180,E1 27274.616,E2 27274.616} C_VEL
LIN {X 0,Y 583.907,Z 775.336,A -85,B 0,C 180,E1 27272.552,E2 27272.552} C_VEL
LIN {X 0,Y 583.898,Z 776.426,A -85,B 0,C 180,E1 27270.392,E2 27270.392} C_VEL
LIN {X 0,Y 583.903,Z 775.887,A -85,B 0,C 180,E1 27268.234,E2 27268.234} C_VEL
LIN {X 0,Y 583.908,Z 773.879,A -85,B 0,C 180,E1 27266.171,E2 27266.171} C_VEL
LIN {X 0,Y 583.915,Z 770.199,A -85,B 0,C 180,E1 27264.103,E2 27264.103} C_VEL
LIN {X 0,Y 583.931,Z 764.682,A -85,B 0,C 180,E1 27261.928,E2 27261.928} C_VEL
LIN {X 0,Y 583.964,Z 757.694,A -85,B 0,C 180,E1 27259.842,E2 27259.842} C_VEL
LIN {X 0,Y 584.006,Z 749.22,A -85,B 0,C 180,E1 27257.843,E2 27257.843} C_VEL
LIN {X 0,Y 584.094,Z 738.983,A -85,B 0,C 180,E1 27255.83,E2 27255.83} C_VEL
LIN {X 0,Y 584.21,Z 727.345,A -85,B 0,C 180,E1 27253.903,E2 27253.903} C_VEL
LIN {X 0,Y 584.352,Z 714.179,A -85,B 0,C 180,E1 27252.053,E2 27252.053} C_VEL
LIN {X 0,Y 584.55,Z 698.891,A -85,B 0,C 180,E1 27250.204,E2 27250.204} C_VEL
LIN {X 0,Y 584.802,Z 682.909,A -85,B 0,C 180,E1 27248.538,E2 27248.538} C_VEL
LIN {X 0,Y 585.083,Z 665.389,A -85,B 0,C 180,E1 27246.962,E2 27246.962} C_VEL
LIN {X 0,Y 585.381,Z 646.412,A -85,B 0,C 180,E1 27245.506,E2 27245.506} C_VEL
LIN {X 0,Y 585.665,Z 627.088,A -85,B 0,C 180,E1 27244.247,E2 27244.247} C_VEL
LIN {X 0,Y 585.992,Z 606.404,A -85,B 0,C 180,E1 27243.117,E2 27243.117} C_VEL
LIN {X 0,Y 586.283,Z 585.909,A -85,B 0,C 180,E1 27242.197,E2 27242.197} C_VEL
LIN {X 0,Y 586.507,Z 564.552,A -85,B 0,C 180,E1 27241.442,E2 27241.442} C_VEL
LIN {X 0,Y 586.742,Z 542.281,A -85,B 0,C 180,E1 27240.853,E2 27240.853} C_VEL
LIN {X 0,Y 586.873,Z 520.449,A -85,B 0,C 180,E1 27240.461,E2 27240.461} C_VEL
LIN {X 0,Y 587.517,Z 292.693,A -85,B 0,C 180,E1 27237.311,E2 27237.311} C_VEL
LIN {X 0,Y 587.515,Z 227.13,A -85,B 0,C 180,E1 27236.374,E2 27236.374} C_VEL
LIN {X 0,Y 587.217,Z 224.044,A -85,B 0,C 180,E1 27236.283,E2 27236.283} C_VEL
LIN {X 0,Y 587.521,Z 176.757,A -85,B 0,C 180,E1 27234.019,E2 27234.019} C_VEL
LIN {X 0,Y 584.266,Z 169.925,A -85,B 0,C 180,E1 27233.449,E2 27233.449} C_VEL
LIN {X 0,Y 584.089,Z 168.981,A -85,B 0,C 180,E1 27233.356,E2 27233.356} C_VEL
LIN {X 0,Y 584.1,Z 169.203,A -85,B 0,C 180,E1 27230.391,E2 27230.391} C_VEL
LIN {X 0,Y 585.257,Z 172.277,A -85,B 0,C 180,E1 27230.255,E2 27230.255} C_VEL
LIN {X 0,Y 587.662,Z 174.693,A -85,B 0,C 180,E1 27229.974,E2 27229.974} C_VEL
LIN {X 0,Y 588.788,Z 175.621,A -85,B 0,C 180,E1 27229.843,E2 27229.843} C_VEL
LIN {X 0,Y 591.538,Z 179.426,A -85,B 0,C 180,E1 27229.529,E2 27229.529} C_VEL
LIN {X 0,Y 593.897,Z 181.83,A -85,B 0,C 180,E1 27229.263,E2 27229.263} C_VEL
LIN {X 0,Y 597.317,Z 185.68,A -85,B 0,C 180,E1 27228.864,E2 27228.864} C_VEL
LIN {X 0,Y 599.93,Z 187.918,A -85,B 0,C 180,E1 27228.382,E2 27228.382} C_VEL
LIN {X 0,Y 601.514,Z 189.006,A -85,B 0,C 180,E1 27227.813,E2 27227.813} C_VEL
LIN {X 0,Y 601.745,Z 189.697,A -85,B 0,C 180,E1 27227.447,E2 27227.447} C_VEL
LIN {X 0,Y 601.061,Z 190.469,A -85,B 0,C 180,E1 27226.909,E2 27226.909} C_VEL
LIN {X 0,Y 599.532,Z 189.808,A -85,B 0,C 180,E1 27226.368,E2 27226.368} C_VEL
LIN {X 0,Y 597.008,Z 187.36,A -85,B 0,C 180,E1 27225.791,E2 27225.791} C_VEL
LIN {X 0,Y 593.411,Z 184.91,A -85,B 0,C 180,E1 27225.319,E2 27225.319} C_VEL
LIN {X 0,Y 589.752,Z 180.787,A -85,B 0,C 180,E1 27224.852,E2 27224.852} C_VEL
LIN {X 0,Y 584.323,Z 170.153,A -85,B 0,C 180,E1 27223.913,E2 27223.913} C_VEL
LIN {X 0,Y 584.094,Z 168.978,A -85,B 0,C 180,E1 27223.828,E2 27223.828} C_VEL
LIN {X 0,Y 584.06,Z 168.979,A -85,B 0,C 180,E1 27220.581,E2 27220.581} C_VEL
LIN {X 0,Y 584.098,Z 168.976,A -85,B 0,C 180,E1 27217.413,E2 27217.413} C_VEL
LIN {X 0,Y 584.055,Z 168.978,A -85,B 0,C 180,E1 27214.222,E2 27214.222} C_VEL
LIN {X 0,Y 584.088,Z 169.135,A -85,B 0,C 180,E1 27210.989,E2 27210.989} C_VEL
LIN {X 0,Y 584.502,Z 176.056,A -85,B 0,C 180,E1 27210.477,E2 27210.477} C_VEL
LIN {X 0,Y 585.118,Z 207.123,A -85,B 0,C 180,E1 27208.085,E2 27208.085} C_VEL
LIN {X 0,Y 585.279,Z 231.537,A -85,B 0,C 180,E1 27206.088,E2 27206.088} C_VEL
LIN {X 0,Y 585.022,Z 267.85,A -85,B 0,C 180,E1 27202.983,E2 27202.983} C_VEL
LIN {X 0,Y 584.748,Z 305.784,A -85,B 0,C 180,E1 27199.789,E2 27199.789} C_VEL
LIN {X 0,Y 584.716,Z 313.084,A -85,B 0,C 180,E1 27199.215,E2 27199.215} C_VEL
LIN {X 0,Y 585.118,Z 319.082,A -85,B 0,C 180,E1 27199.124,E2 27199.124} C_VEL
LIN {X 0,Y 584.863,Z 481.919,A -85,B 0,C 180,E1 27197.045,E2 27197.045} C_VEL
LIN {X 0,Y 584.808,Z 499.579,A -85,B 0,C 180,E1 27196.635,E2 27196.635} C_VEL
LIN {X 0,Y 584.705,Z 516.653,A -85,B 0,C 180,E1 27196.046,E2 27196.046} C_VEL
LIN {X 0,Y 584.571,Z 533.246,A -85,B 0,C 180,E1 27195.272,E2 27195.272} C_VEL
LIN {X 0,Y 584.436,Z 548.429,A -85,B 0,C 180,E1 27194.363,E2 27194.363} C_VEL
LIN {X 0,Y 584.297,Z 562.616,A -85,B 0,C 180,E1 27193.306,E2 27193.306} C_VEL
LIN {X 0,Y 584.181,Z 576.333,A -85,B 0,C 180,E1 27192.052,E2 27192.052} C_VEL
LIN {X 0,Y 584.084,Z 588.317,A -85,B 0,C 180,E1 27190.703,E2 27190.703} C_VEL
LIN {X 0,Y 584.007,Z 598.705,A -85,B 0,C 180,E1 27189.261,E2 27189.261} C_VEL
LIN {X 0,Y 583.961,Z 607.853,A -85,B 0,C 180,E1 27187.675,E2 27187.675} C_VEL
LIN {X 0,Y 583.934,Z 614.942,A -85,B 0,C 180,E1 27186.094,E2 27186.094} C_VEL
LIN {X 0,Y 583.922,Z 620.468,A -85,B 0,C 180,E1 27184.419,E2 27184.419} C_VEL
LIN {X 0,Y 583.914,Z 624.141,A -85,B 0,C 180,E1 27182.748,E2 27182.748} C_VEL
LIN {X 0,Y 583.911,Z 626.161,A -85,B 0,C 180,E1 27180.981,E2 27180.981} C_VEL
LIN {X 0,Y 583.914,Z 626.334,A -85,B 0,C 180,E1 27179.215,E2 27179.215} C_VEL
LIN {X 0,Y 583.915,Z 624.6,A -85,B 0,C 180,E1 27177.448,E2 27177.448} C_VEL
LIN {X 0,Y 583.918,Z 620.948,A -85,B 0,C 180,E1 27175.679,E2 27175.679} C_VEL
LIN {X 0,Y 583.929,Z 615.651,A -85,B 0,C 180,E1 27174.004,E2 27174.004} C_VEL
LIN {X 0,Y 583.961,Z 608.817,A -85,B 0,C 180,E1 27172.424,E2 27172.424} C_VEL
LIN {X 0,Y 584.003,Z 599.921,A -85,B 0,C 180,E1 27170.838,E2 27170.838} C_VEL
LIN {X 0,Y 584.07,Z 589.386,A -85,B 0,C 180,E1 27169.345,E2 27169.345} C_VEL
